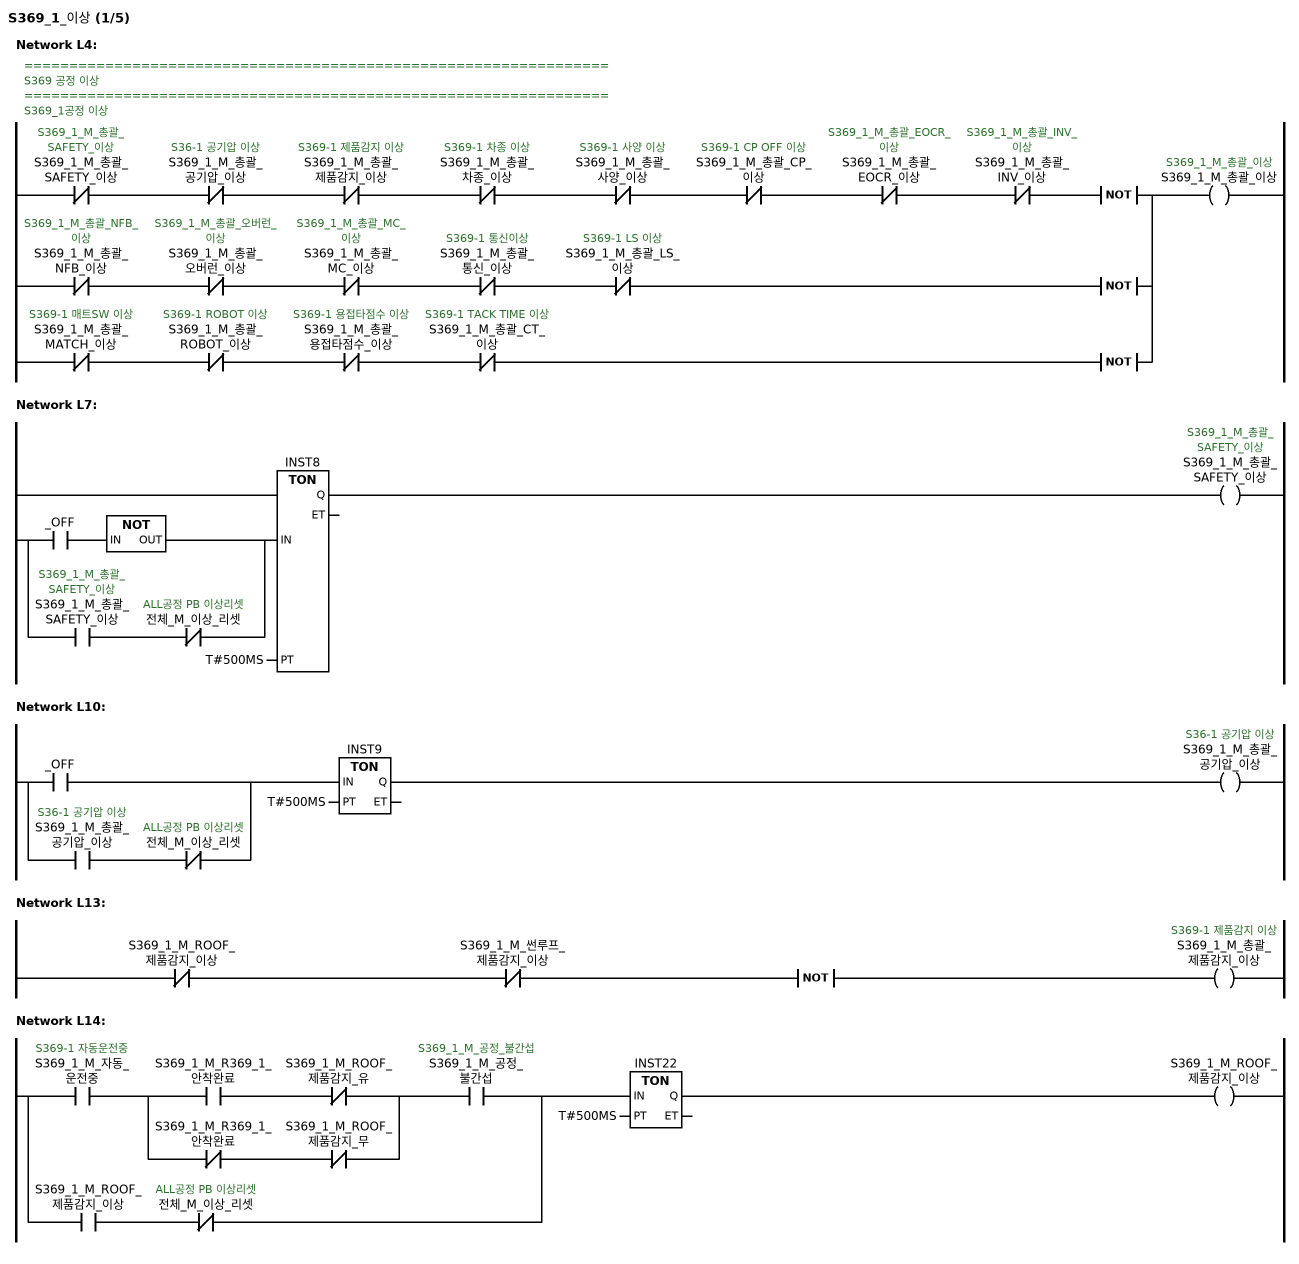
(* [picture p264: S369_1_이상 rungs L4-L14] *)
(* ================================================================= *)
(* S369 공정 이상 *)
(* ================================================================= *)
(* S369_1공정 이상 *)
(* Rung L4 *)
S369_1_M_총괄_이상 := NOT (NOT S369_1_M_총괄_SAFETY_이상 AND NOT S369_1_M_총괄_공기압_이상 AND NOT S369_1_M_총괄_제품감지_이상 AND NOT S369_1_M_총괄_차종_이상 AND NOT S369_1_M_총괄_사양_이상 AND NOT S369_1_M_총괄_CP_이상 AND NOT S369_1_M_총괄_EOCR_이상 AND NOT S369_1_M_총괄_INV_이상) OR NOT (NOT S369_1_M_총괄_NFB_이상 AND NOT S369_1_M_총괄_오버런_이상 AND NOT S369_1_M_총괄_MC_이상 AND NOT S369_1_M_총괄_통신_이상 AND NOT S369_1_M_총괄_LS_이상) OR NOT (NOT S369_1_M_총괄_MATCH_이상 AND NOT S369_1_M_총괄_ROBOT_이상 AND NOT S369_1_M_총괄_용접타점수_이상 AND NOT S369_1_M_총괄_CT_이상);
(* Rung L7 *)
INST8(IN := (NOT _OFF) OR (S369_1_M_총괄_SAFETY_이상 AND NOT 전체_M_이상_리셋), PT := T#500MS);
S369_1_M_총괄_SAFETY_이상 := INST8.Q;
(* Rung L10 *)
INST9(IN := _OFF OR (S369_1_M_총괄_공기압_이상 AND NOT 전체_M_이상_리셋), PT := T#500MS);
S369_1_M_총괄_공기압_이상 := INST9.Q;
(* Rung L13 *)
S369_1_M_총괄_제품감지_이상 := NOT (NOT S369_1_M_ROOF_제품감지_이상 AND NOT S369_1_M_썬루프_제품감지_이상);
(* Rung L14 *)
INST22(IN := (S369_1_M_자동_운전중 AND ((S369_1_M_R369_1_안착완료 AND NOT S369_1_M_ROOF_제품감지_유) OR (NOT S369_1_M_R369_1_안착완료 AND NOT S369_1_M_ROOF_제품감지_무)) AND S369_1_M_공정_불간섭) OR (S369_1_M_ROOF_제품감지_이상 AND NOT 전체_M_이상_리셋), PT := T#500MS);
S369_1_M_ROOF_제품감지_이상 := INST22.Q;

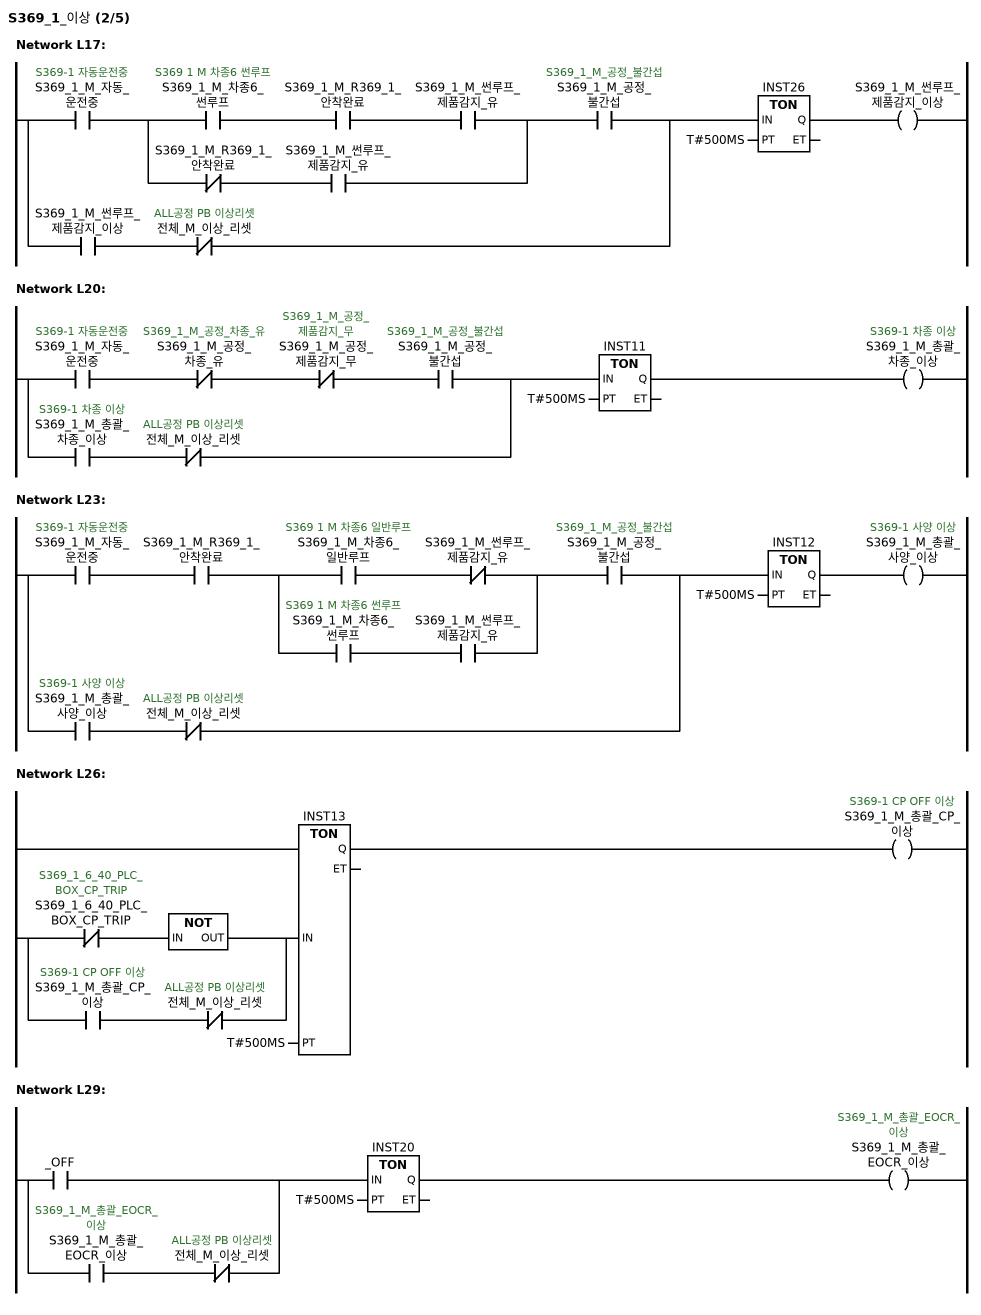
(* Rung L17 *)
INST26(IN := (S369_1_M_자동_운전중 AND ((S369_1_M_차종6_썬루프 AND S369_1_M_R369_1_안착완료 AND S369_1_M_썬루프_제품감지_유) OR (NOT S369_1_M_R369_1_안착완료 AND S369_1_M_썬루프_제품감지_유)) AND S369_1_M_공정_불간섭) OR (S369_1_M_썬루프_제품감지_이상 AND NOT 전체_M_이상_리셋), PT := T#500MS);
S369_1_M_썬루프_제품감지_이상 := INST26.Q;
(* Rung L20 *)
INST11(IN := (S369_1_M_자동_운전중 AND NOT S369_1_M_공정_차종_유 AND NOT S369_1_M_공정_제품감지_무 AND S369_1_M_공정_불간섭) OR (S369_1_M_총괄_차종_이상 AND NOT 전체_M_이상_리셋), PT := T#500MS);
S369_1_M_총괄_차종_이상 := INST11.Q;
(* Rung L23 *)
INST12(IN := (S369_1_M_자동_운전중 AND S369_1_M_R369_1_안착완료 AND ((S369_1_M_차종6_일반루프 AND NOT S369_1_M_썬루프_제품감지_유) OR (S369_1_M_차종6_썬루프 AND S369_1_M_썬루프_제품감지_유)) AND S369_1_M_공정_불간섭) OR (S369_1_M_총괄_사양_이상 AND NOT 전체_M_이상_리셋), PT := T#500MS);
S369_1_M_총괄_사양_이상 := INST12.Q;
(* Rung L26 *)
INST13(IN := (NOT (NOT S369_1_6_40_PLC_BOX_CP_TRIP)) OR (S369_1_M_총괄_CP_이상 AND NOT 전체_M_이상_리셋), PT := T#500MS);
S369_1_M_총괄_CP_이상 := INST13.Q;
(* Rung L29 *)
INST20(IN := _OFF OR (S369_1_M_총괄_EOCR_이상 AND NOT 전체_M_이상_리셋), PT := T#500MS);
S369_1_M_총괄_EOCR_이상 := INST20.Q;

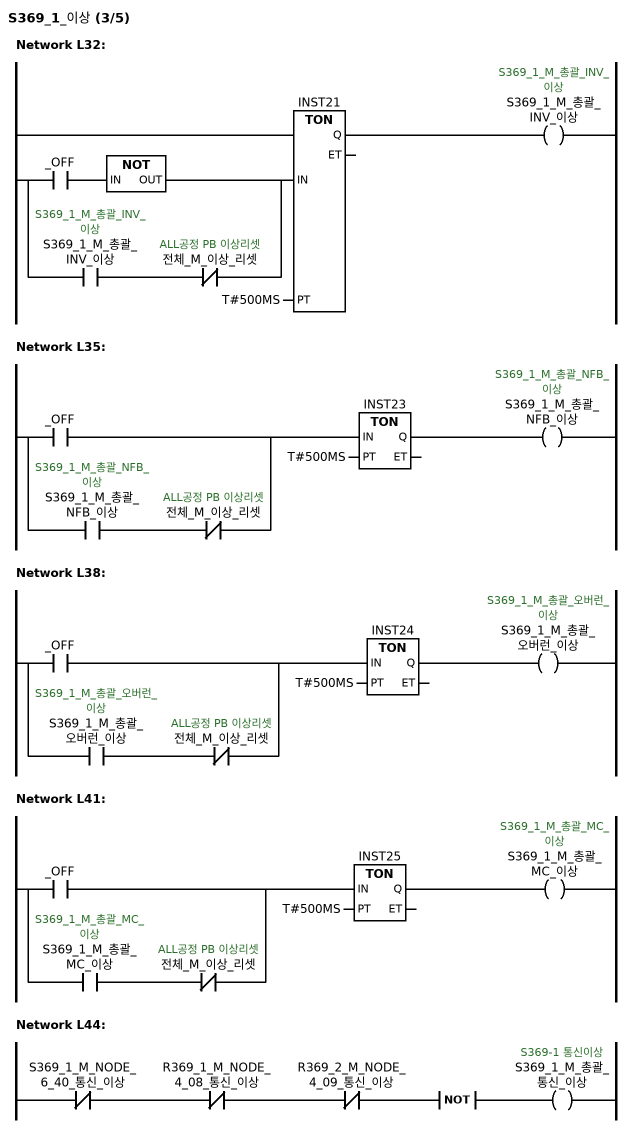
(* Rung L32 *)
INST21(IN := (NOT _OFF) OR (S369_1_M_총괄_INV_이상 AND NOT 전체_M_이상_리셋), PT := T#500MS);
S369_1_M_총괄_INV_이상 := INST21.Q;
(* Rung L35 *)
INST23(IN := _OFF OR (S369_1_M_총괄_NFB_이상 AND NOT 전체_M_이상_리셋), PT := T#500MS);
S369_1_M_총괄_NFB_이상 := INST23.Q;
(* Rung L38 *)
INST24(IN := _OFF OR (S369_1_M_총괄_오버런_이상 AND NOT 전체_M_이상_리셋), PT := T#500MS);
S369_1_M_총괄_오버런_이상 := INST24.Q;
(* Rung L41 *)
INST25(IN := _OFF OR (S369_1_M_총괄_MC_이상 AND NOT 전체_M_이상_리셋), PT := T#500MS);
S369_1_M_총괄_MC_이상 := INST25.Q;
(* Rung L44 *)
S369_1_M_총괄_통신_이상 := NOT (NOT S369_1_M_NODE_6_40_통신_이상 AND NOT R369_1_M_NODE_4_08_통신_이상 AND NOT R369_2_M_NODE_4_09_통신_이상);

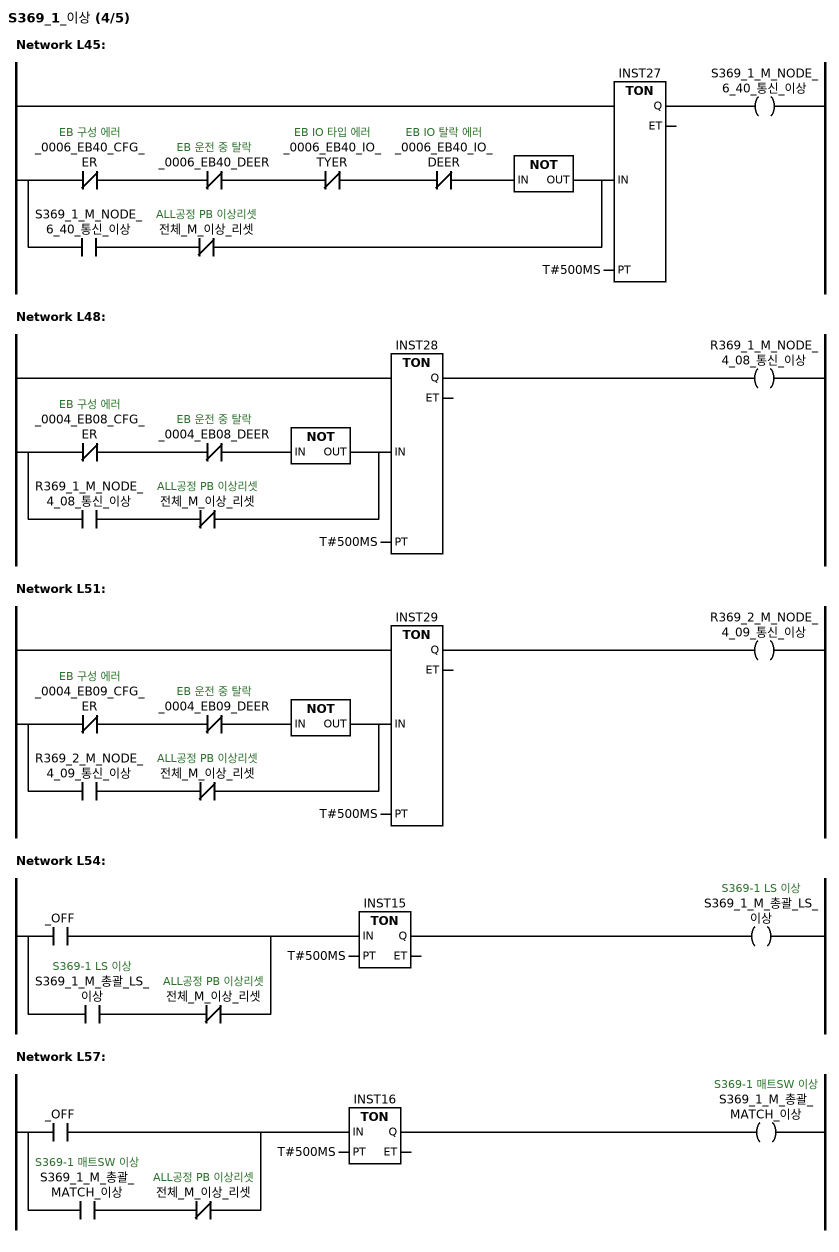
(* Rung L45 *)
INST27(IN := (NOT (NOT _0006_EB40_CFG_ER AND NOT _0006_EB40_DEER AND NOT _0006_EB40_IO_TYER AND NOT _0006_EB40_IO_DEER)) OR (S369_1_M_NODE_6_40_통신_이상 AND NOT 전체_M_이상_리셋), PT := T#500MS);
S369_1_M_NODE_6_40_통신_이상 := INST27.Q;
(* Rung L48 *)
INST28(IN := (NOT (NOT _0004_EB08_CFG_ER AND NOT _0004_EB08_DEER)) OR (R369_1_M_NODE_4_08_통신_이상 AND NOT 전체_M_이상_리셋), PT := T#500MS);
R369_1_M_NODE_4_08_통신_이상 := INST28.Q;
(* Rung L51 *)
INST29(IN := (NOT (NOT _0004_EB09_CFG_ER AND NOT _0004_EB09_DEER)) OR (R369_2_M_NODE_4_09_통신_이상 AND NOT 전체_M_이상_리셋), PT := T#500MS);
R369_2_M_NODE_4_09_통신_이상 := INST29.Q;
(* Rung L54 *)
INST15(IN := _OFF OR (S369_1_M_총괄_LS_이상 AND NOT 전체_M_이상_리셋), PT := T#500MS);
S369_1_M_총괄_LS_이상 := INST15.Q;
(* Rung L57 *)
INST16(IN := _OFF OR (S369_1_M_총괄_MATCH_이상 AND NOT 전체_M_이상_리셋), PT := T#500MS);
S369_1_M_총괄_MATCH_이상 := INST16.Q;

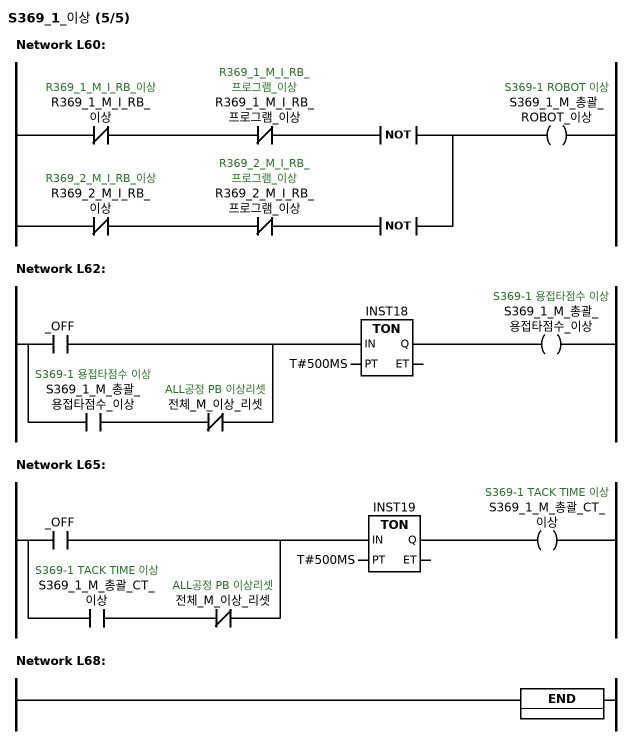
(* Rung L60 *)
S369_1_M_총괄_ROBOT_이상 := NOT (NOT R369_1_M_I_RB_이상 AND NOT R369_1_M_I_RB_프로그램_이상) OR NOT (NOT R369_2_M_I_RB_이상 AND NOT R369_2_M_I_RB_프로그램_이상);
(* Rung L62 *)
INST18(IN := _OFF OR (S369_1_M_총괄_용접타점수_이상 AND NOT 전체_M_이상_리셋), PT := T#500MS);
S369_1_M_총괄_용접타점수_이상 := INST18.Q;
(* Rung L65 *)
INST19(IN := _OFF OR (S369_1_M_총괄_CT_이상 AND NOT 전체_M_이상_리셋), PT := T#500MS);
S369_1_M_총괄_CT_이상 := INST19.Q;
(* Rung L68 *)
END();
END_PROGRAM

PROGRAM S369_유틸리티 (* task: 스캔 프로그램 *)
VAR_EXTERNAL RETAIN
    ALWAYS_OFF : BOOL; (* AT %MW3.0 *) (* 항시 OFF *)
    HMI_M_선택_MOD_S368 : BOOL; (* AT %MW6.6 *) (* HMI M 선택 MOD S368 *)
    HMI_M_선택_MOD_S369_LD : BOOL; (* AT %MW6.8 *) (* HMI M 선택 MOD S369 *)
    HMI_M_선택_MOD_S369_UD : BOOL; (* AT %MW6.9 *)
    S368_M_공정_제품감지_무 : BOOL; (* AT %MW4001.6 *) (* S368_M_공정_제품감지_무 *)
    S368_M_공정_차종_무 : BOOL; (* AT %MW4002.1 *) (* S368_M_공정_차종_무 *)
    S368_M_작업완료_SET_PLS : BOOL; (* AT %MW4000.8 *) (* S368 M 작업완료 SET PLS *)
    S368_M_작업완료_리셋_PLS : BOOL; (* AT %MW4000.9 *) (* S368 M 작업완료 리셋 PLS *)
    S369_1_M_공정_차종_무 : BOOL; (* AT %MW4502.1 *) (* S369_1_M_공정_차종_무 *)
    S369_1_M_공정_차종_유 : BOOL; (* AT %MW4502.0 *) (* S369_1_M_공정_차종_유 *)
    S369_1_M_총괄_이상 : BOOL; (* AT %MW4509.0 *) (* S369_1_M_총괄_이상 *)
    S369_M_LD_BYPASS_보조 : BOOL; (* AT %MW5003.14 *)
    S369_M_LD_EJECT_상승단 : BOOL; (* AT %MW5100.3 *) (* S369_M_LD_EJECT_상승단 *)
    S369_M_LD_EJECT_하강단 : BOOL; (* AT %MW5100.4 *) (* S369_M_LD_EJECT_하강단 *)
    S369_M_LD_LH_LAT_전진단 : BOOL; (* AT %MW5101.3 *) (* S369_M_LD_LH_LAT_전진단 *)
    S369_M_LD_LH_LAT_후진단 : BOOL; (* AT %MW5101.4 *) (* S369_M_LD_LH_LAT_후진단 *)
    S369_M_LD_RH_LAT_전진단 : BOOL; (* AT %MW5102.3 *) (* S369_M_LD_RH_LAT_전진단 *)
    S369_M_LD_RH_LAT_후진단 : BOOL; (* AT %MW5102.4 *) (* S369_M_LD_RH_LAT_후진단 *)
    S369_M_LD_작업완료_SET_PLS : BOOL; (* AT %MW5000.6 *)
    S369_M_LD_작업완료_리셋_PLS : BOOL; (* AT %MW5000.7 *)
    S369_M_R308_3_언로딩가능 : BOOL; (* AT %MW5004.9 *)
    S369_M_R308_3_언로딩완료 : BOOL; (* AT %MW5001.5 *)
    S369_M_R308_3_클램프완료 : BOOL; (* AT %MW5001.4 *)
    S369_M_R308_3_클램프요구 : BOOL; (* AT %MW5004.11 *)
    S369_M_R308_3_행거안착가능 : BOOL; (* AT %MW5004.10 *)
    S369_M_R308_3_행거안착완료 : BOOL; (* AT %MW5001.3 *)
    S369_M_R369_2_로딩가능 : BOOL; (* AT %MW5004.8 *)
    S369_M_R369_2_로딩완료 : BOOL; (* AT %MW5001.2 *)
    S369_M_UD_BYPASS_보조 : BOOL; (* AT %MW5003.15 *) (* S369 M BYPASS 보조 *)
    S369_M_UD_DOCK_CLP_전진단 : BOOL; (* AT %MW5111.3 *) (* S369_M_UD_DOCK_CLP_전진단 *)
    S369_M_UD_DOCK_CLP_후진단 : BOOL; (* AT %MW5111.4 *) (* S369_M_UD_DOCK_CLP_후진단 *)
    S369_M_UD_EJECT_상승단 : BOOL; (* AT %MW5108.3 *) (* S369_M_UD_EJECT_상승단 *)
    S369_M_UD_EJECT_하강단 : BOOL; (* AT %MW5108.4 *) (* S369_M_UD_EJECT_하강단 *)
    S369_M_UD_LH_LAT_전진단 : BOOL; (* AT %MW5109.3 *) (* S369_M_UD_LH_LAT_전진단 *)
    S369_M_UD_LH_LAT_후진단 : BOOL; (* AT %MW5109.4 *) (* S369_M_UD_LH_LAT_후진단 *)
    S369_M_UD_RH_LAT_전진단 : BOOL; (* AT %MW5110.3 *) (* S369_M_UD_RH_LAT_전진단 *)
    S369_M_UD_RH_LAT_후진단 : BOOL; (* AT %MW5110.4 *) (* S369_M_UD_RH_LAT_후진단 *)
    S369_M_UD_작업완료_SET_PLS : BOOL; (* AT %MW5000.8 *) (* S369 M 작업완료 SET PLS *)
    S369_M_UD_작업완료_리셋_PLS : BOOL; (* AT %MW5000.9 *) (* S369 M 작업완료 리셋 PLS *)
    S369_M_로딩_공정_불간섭 : BOOL; (* AT %MW5004.2 *) (* S369_M_공정_불간섭 *)
    S369_M_로딩_공정_원위치 : BOOL; (* AT %MW5004.0 *) (* S369_M_공정_원위치 *)
    S369_M_로딩_리셋보조 : BOOL; (* AT %MW5000.13 *)
    S369_M_로딩_이젝터_제품감지_무 : BOOL; (* AT %MW5001.9 *)
    S369_M_로딩_이젝터_제품감지_유 : BOOL; (* AT %MW5001.8 *)
    S369_M_로딩_작업_완료 : BOOL; (* AT %MW5001.0 *) (* S369_M_작업_완료 *)
    S369_M_로딩버퍼_SEQ : WORD; (* AT %MW10240 *) (* S369 M 로딩버퍼 SEQ *)
    S369_M_로딩버퍼_제품감지_무 : BOOL; (* AT %MW5005.1 *) (* S369_로딩버퍼_제품감지_무 *)
    S369_M_로딩버퍼_제품감지_유 : BOOL; (* AT %MW5005.0 *) (* S369_로딩버퍼_제품감지_유 *)
    S369_M_로딩버퍼_차종1_AX : BOOL; (* AT %MW10241.0 *) (* S369 M 로딩버퍼 차종1 AX *)
    S369_M_로딩버퍼_차종1_B : BOOL; (* AT %MW10241.1 *) (* S369 M 로딩버퍼 차종1 B *)
    S369_M_로딩버퍼_차종1_C : BOOL; (* AT %MW10241.2 *) (* S369 M 로딩버퍼 차종1 C *)
    S369_M_로딩버퍼_차종1_D : BOOL; (* AT %MW10241.3 *) (* S369 M 로딩버퍼 차종1 D *)
    S369_M_로딩버퍼_차종1_E : BOOL; (* AT %MW10241.4 *) (* S369 M 로딩버퍼 차종1 E *)
    S369_M_로딩버퍼_차종1_F : BOOL; (* AT %MW10241.5 *) (* S369 M 로딩버퍼 차종1 F *)
    S369_M_로딩버퍼_차종1_G : BOOL; (* AT %MW10241.6 *) (* S369 M 로딩버퍼 차종1 G *)
    S369_M_로딩버퍼_차종1_H : BOOL; (* AT %MW10241.7 *) (* S369 M 로딩버퍼 차종1 H *)
    S369_M_로딩버퍼_차종2_3DR : BOOL; (* AT %MW10241.8 *) (* S369 M 로딩버퍼 차종2 3DR *)
    S369_M_로딩버퍼_차종2_4DR : BOOL; (* AT %MW10241.9 *) (* S369 M 로딩버퍼 차종2 4DR *)
    S369_M_로딩버퍼_차종2_5DR : BOOL; (* AT %MW10241.10 *) (* S369 M 로딩버퍼 차종2 5DR *)
    S369_M_로딩버퍼_차종2_SP1 : BOOL; (* AT %MW10241.12 *) (* S369 M 로딩버퍼 차종2 SP1 *)
    S369_M_로딩버퍼_차종2_SP2 : BOOL; (* AT %MW10241.13 *) (* S369 M 로딩버퍼 차종2 SP2 *)
    S369_M_로딩버퍼_차종2_WGN : BOOL; (* AT %MW10241.11 *) (* S369 M 로딩버퍼 차종2 WGN *)
    S369_M_로딩버퍼_차종3_LHD : BOOL; (* AT %MW10241.14 *) (* S369 M 로딩버퍼 차종3 LHD *)
    S369_M_로딩버퍼_차종3_RHD : BOOL; (* AT %MW10241.15 *) (* S369 M 로딩버퍼 차종3 RHD *)
    S369_M_로딩버퍼_차종4_EEC : BOOL; (* AT %MW10242.3 *) (* S369 M 로딩버퍼 차종4 EEC *)
    S369_M_로딩버퍼_차종4_SP1 : BOOL; (* AT %MW10242.8 *) (* S369 M 로딩버퍼 차종4 SP1 *)
    S369_M_로딩버퍼_차종4_SP2 : BOOL; (* AT %MW10242.9 *) (* S369 M 로딩버퍼 차종4 SP2 *)
    S369_M_로딩버퍼_차종4_SP3 : BOOL; (* AT %MW10242.11 *) (* S369 M 로딩버퍼 차종4 SP3 *)
    S369_M_로딩버퍼_차종4_SP4 : BOOL; (* AT %MW10242.12 *) (* S369 M 로딩버퍼 차종4 SP4 *)
    S369_M_로딩버퍼_차종4_SP5 : BOOL; (* AT %MW10242.13 *) (* S369 M 로딩버퍼 차종4 SP5 *)
    S369_M_로딩버퍼_차종4_SP6 : BOOL; (* AT %MW10242.14 *) (* S369 M 로딩버퍼 차종4 SP6 *)
    S369_M_로딩버퍼_차종4_SP7 : BOOL; (* AT %MW10242.15 *) (* S369 M 로딩버퍼 차종4 SP7 *)
    S369_M_로딩버퍼_차종4_내수 : BOOL; (* AT %MW10242.0 *) (* S369 M 로딩버퍼 차종4 내수 *)
    S369_M_로딩버퍼_차종4_러시아 : BOOL; (* AT %MW10242.10 *) (* S369 M 로딩버퍼 차종4 러시아 *)
    S369_M_로딩버퍼_차종4_북미 : BOOL; (* AT %MW10242.2 *) (* S369 M 로딩버퍼 차종4 북미 *)
    S369_M_로딩버퍼_차종4_브라질 : BOOL; (* AT %MW10242.7 *) (* S369 M 로딩버퍼 차종4 브라질 *)
    S369_M_로딩버퍼_차종4_수출 : BOOL; (* AT %MW10242.1 *) (* S369 M 로딩버퍼 차종4 수출 *)
    S369_M_로딩버퍼_차종4_중국 : BOOL; (* AT %MW10242.6 *) (* S369 M 로딩버퍼 차종4 중국 *)
    S369_M_로딩버퍼_차종4_중동 : BOOL; (* AT %MW10242.5 *) (* S369 M 로딩버퍼 차종4 중동 *)
    S369_M_로딩버퍼_차종4_호주 : BOOL; (* AT %MW10242.4 *) (* S369 M 로딩버퍼 차종4 호주 *)
    S369_M_로딩버퍼_차종5_AT : BOOL; (* AT %MW10243.1 *) (* S369 M 로딩버퍼 차종5 AT *)
    S369_M_로딩버퍼_차종5_MT : BOOL; (* AT %MW10243.0 *) (* S369 M 로딩버퍼 차종5 MT *)
    S369_M_로딩버퍼_차종5_SP1 : BOOL; (* AT %MW10243.2 *) (* S369 M 로딩버퍼 차종5 SP1 *)
    S369_M_로딩버퍼_차종6_DSROOF : BOOL; (* AT %MW10243.6 *) (* S369 M 로딩버퍼 차종6 DSROOF *)
    S369_M_로딩버퍼_차종6_SP1 : BOOL; (* AT %MW10243.7 *) (* S369 M 로딩버퍼 차종6 SP1 *)
    S369_M_로딩버퍼_차종6_썬루프 : BOOL; (* AT %MW10243.4 *) (* S369 M 로딩버퍼 차종6 썬루프 *)
    S369_M_로딩버퍼_차종6_일반루프 : BOOL; (* AT %MW10243.3 *) (* S369 M 로딩버퍼 차종6 일반루프 *)
    S369_M_로딩버퍼_차종6_파노라마루프 : BOOL; (* AT %MW10243.5 *) (* S369 M 로딩버퍼 차종6 파노라마루프 *)
    S369_M_로딩버퍼_차종7_DSL : BOOL; (* AT %MW10243.9 *) (* S369 M 로딩버퍼 차종7 DSL *)
    S369_M_로딩버퍼_차종7_GSL : BOOL; (* AT %MW10243.8 *) (* S369 M 로딩버퍼 차종7 GSL *)
    S369_M_로딩버퍼_차종7_SP1 : BOOL; (* AT %MW10243.10 *) (* S369 M 로딩버퍼 차종7 SP1 *)
    S369_M_로딩버퍼_차종7_SP2 : BOOL; (* AT %MW10243.11 *) (* S369 M 로딩버퍼 차종7 SP2 *)
    S369_M_로딩버퍼_차종7_SP3 : BOOL; (* AT %MW10243.12 *) (* S369 M 로딩버퍼 차종7 SP3 *)
    S369_M_로딩버퍼_차종7_SP4 : BOOL; (* AT %MW10243.13 *) (* S369 M 로딩버퍼 차종7 SP4 *)
    S369_M_로딩버퍼_차종7_SP5 : BOOL; (* AT %MW10243.14 *) (* S369 M 로딩버퍼 차종7 SP5 *)
    S369_M_로딩버퍼_차종7_SP6 : BOOL; (* AT %MW10243.15 *) (* S369 M 로딩버퍼 차종7 SP6 *)
    S369_M_로딩버퍼_차종8_2WD : BOOL; (* AT %MW10244.0 *) (* S369 M 로딩버퍼 차종8 2WD *)
    S369_M_로딩버퍼_차종8_4WD : BOOL; (* AT %MW10244.1 *) (* S369 M 로딩버퍼 차종8 4WD *)
    S369_M_로딩버퍼_차종8_SP1 : BOOL; (* AT %MW10244.2 *) (* S369 M 로딩버퍼 차종8 SP1 *)
    S369_M_로딩버퍼_차종9_MPI : BOOL; (* AT %MW10244.3 *) (* S369 M 로딩버퍼 차종9 MPI *)
    S369_M_로딩버퍼_차종9_SP1 : BOOL; (* AT %MW10244.5 *) (* S369 M 로딩버퍼 차종9 SP1 *)
    S369_M_로딩버퍼_차종9_SP10 : BOOL; (* AT %MW10244.14 *) (* S369 M 로딩버퍼 차종9 SP10 *)
    S369_M_로딩버퍼_차종9_SP11 : BOOL; (* AT %MW10244.15 *) (* S369 M 로딩버퍼 차종9 SP11 *)
    S369_M_로딩버퍼_차종9_SP2 : BOOL; (* AT %MW10244.6 *) (* S369 M 로딩버퍼 차종9 SP2 *)
    S369_M_로딩버퍼_차종9_SP3 : BOOL; (* AT %MW10244.7 *) (* S369 M 로딩버퍼 차종9 SP3 *)
    S369_M_로딩버퍼_차종9_SP4 : BOOL; (* AT %MW10244.8 *) (* S369 M 로딩버퍼 차종9 SP4 *)
    S369_M_로딩버퍼_차종9_SP5 : BOOL; (* AT %MW10244.9 *) (* S369 M 로딩버퍼 차종9 SP5 *)
    S369_M_로딩버퍼_차종9_SP6 : BOOL; (* AT %MW10244.10 *) (* S369 M 로딩버퍼 차종9 SP6 *)
    S369_M_로딩버퍼_차종9_SP7 : BOOL; (* AT %MW10244.11 *) (* S369 M 로딩버퍼 차종9 SP7 *)
    S369_M_로딩버퍼_차종9_SP8 : BOOL; (* AT %MW10244.12 *) (* S369 M 로딩버퍼 차종9 SP8 *)
    S369_M_로딩버퍼_차종9_SP9 : BOOL; (* AT %MW10244.13 *) (* S369 M 로딩버퍼 차종9 SP9 *)
    S369_M_로딩버퍼_차종9_T_GDI : BOOL; (* AT %MW10244.4 *) (* S369 M 로딩버퍼 차종9 T GDI *)
    S369_M_로딩버퍼_차종_OPT1_R_RACK_무 : BOOL; (* AT %MW10245.3 *) (* S369 M 로딩버퍼 차종 OPT1 R RACK 무 *)
    S369_M_로딩버퍼_차종_OPT1_R_RACK_유 : BOOL; (* AT %MW10245.2 *) (* S369 M 로딩버퍼 차종 OPT1 R RACK 유 *)
    S369_M_로딩버퍼_차종_OPT1_S_REP_EATER_무 : BOOL; (* AT %MW10245.7 *) (* S369 M 로딩버퍼 차종 OPT1 S REP EATER 무 *)
    S369_M_로딩버퍼_차종_OPT1_S_REP_EATER_유 : BOOL; (* AT %MW10245.6 *) (* S369 M 로딩버퍼 차종 OPT1 S REP EATER 유 *)
    S369_M_로딩버퍼_차종_OPT1_VAN_무 : BOOL; (* AT %MW10245.9 *) (* S369 M 로딩버퍼 차종 OPT1 VAN 무 *)
    S369_M_로딩버퍼_차종_OPT1_VAN_유 : BOOL; (* AT %MW10245.8 *) (* S369 M 로딩버퍼 차종 OPT1 VAN 유 *)
    S369_M_로딩버퍼_차종_OPT1_슬라이딩_무 : BOOL; (* AT %MW10245.1 *) (* S369 M 로딩버퍼 차종 OPT1 슬라이딩 무 *)
    S369_M_로딩버퍼_차종_OPT1_슬라이딩_유 : BOOL; (* AT %MW10245.0 *) (* S369 M 로딩버퍼 차종 OPT1 슬라이딩 유 *)
    S369_M_로딩버퍼_차종_OPT1_폴딩_무 : BOOL; (* AT %MW10245.5 *) (* S369 M 로딩버퍼 차종 OPT1 폴딩 무 *)
    S369_M_로딩버퍼_차종_OPT1_폴딩_유 : BOOL; (* AT %MW10245.4 *) (* S369 M 로딩버퍼 차종 OPT1 폴딩 유 *)
    S369_M_로딩버퍼_차종_공대차 : BOOL; (* AT %MW10250.12 *) (* S369 M 로딩버퍼 차종 공대차 *)
    S369_M_로딩버퍼_차종_공차 : BOOL; (* AT %MW10250.10 *) (* S369 M 로딩버퍼 차종 공차 *)
    S369_M_로딩버퍼_차종_무 : BOOL; (* AT %MW5002.1 *)
    S369_M_로딩버퍼_차종_불량차 : BOOL; (* AT %MW10250.11 *) (* S369 M 로딩버퍼 차종 불량차 *)
    S369_M_로딩버퍼_차종_유 : BOOL; (* AT %MW5002.0 *)
    S369_M_수동모드 : BOOL; (* AT %MW5000.3 *) (* S369 선택 수동모드 *)
    S369_M_언로딩_공정_불간섭 : BOOL; (* AT %MW5004.3 *)
    S369_M_언로딩_공정_원위치 : BOOL; (* AT %MW5004.1 *)
    S369_M_언로딩_이젝터_제품감지_무 : BOOL; (* AT %MW5001.11 *)
    S369_M_언로딩_이젝터_제품감지_유 : BOOL; (* AT %MW5001.10 *)
    S369_M_언로딩_작업_완료 : BOOL; (* AT %MW5001.1 *)
    S369_M_언로딩버퍼_SEQ : WORD; (* AT %MW10340 *) (* S369 M 언로딩버퍼 SEQ *)
    S369_M_언로딩버퍼_제품감지_무 : BOOL; (* AT %MW5005.11 *) (* S369_언로딩버퍼_제품감지_무 *)
    S369_M_언로딩버퍼_제품감지_유 : BOOL; (* AT %MW5005.10 *) (* S369_언로딩버퍼_제품감지_유 *)
    S369_M_언로딩버퍼_차종1_AX : BOOL; (* AT %MW10341.0 *) (* S369 M 언로딩버퍼 차종1 AX *)
    S369_M_언로딩버퍼_차종1_B : BOOL; (* AT %MW10341.1 *) (* S369 M 언로딩버퍼 차종1 B *)
    S369_M_언로딩버퍼_차종1_C : BOOL; (* AT %MW10341.2 *) (* S369 M 언로딩버퍼 차종1 C *)
    S369_M_언로딩버퍼_차종1_D : BOOL; (* AT %MW10341.3 *) (* S369 M 언로딩버퍼 차종1 D *)
    S369_M_언로딩버퍼_차종1_E : BOOL; (* AT %MW10341.4 *) (* S369 M 언로딩버퍼 차종1 E *)
    S369_M_언로딩버퍼_차종1_F : BOOL; (* AT %MW10341.5 *) (* S369 M 언로딩버퍼 차종1 F *)
    S369_M_언로딩버퍼_차종1_G : BOOL; (* AT %MW10341.6 *) (* S369 M 언로딩버퍼 차종1 G *)
    S369_M_언로딩버퍼_차종1_H : BOOL; (* AT %MW10341.7 *) (* S369 M 언로딩버퍼 차종1 H *)
    S369_M_언로딩버퍼_차종2_3DR : BOOL; (* AT %MW10341.8 *) (* S369 M 언로딩버퍼 차종2 3DR *)
    S369_M_언로딩버퍼_차종2_4DR : BOOL; (* AT %MW10341.9 *) (* S369 M 언로딩버퍼 차종2 4DR *)
    S369_M_언로딩버퍼_차종2_5DR : BOOL; (* AT %MW10341.10 *) (* S369 M 언로딩버퍼 차종2 5DR *)
    S369_M_언로딩버퍼_차종2_SP1 : BOOL; (* AT %MW10341.12 *) (* S369 M 언로딩버퍼 차종2 SP1 *)
    S369_M_언로딩버퍼_차종2_SP2 : BOOL; (* AT %MW10341.13 *) (* S369 M 언로딩버퍼 차종2 SP2 *)
    S369_M_언로딩버퍼_차종2_WGN : BOOL; (* AT %MW10341.11 *) (* S369 M 언로딩버퍼 차종2 WGN *)
    S369_M_언로딩버퍼_차종3_LHD : BOOL; (* AT %MW10341.14 *) (* S369 M 언로딩버퍼 차종3 LHD *)
    S369_M_언로딩버퍼_차종3_RHD : BOOL; (* AT %MW10341.15 *) (* S369 M 언로딩버퍼 차종3 RHD *)
    S369_M_언로딩버퍼_차종4_EEC : BOOL; (* AT %MW10342.3 *) (* S369 M 언로딩버퍼 차종4 EEC *)
    S369_M_언로딩버퍼_차종4_SP1 : BOOL; (* AT %MW10342.8 *) (* S369 M 언로딩버퍼 차종4 SP1 *)
    S369_M_언로딩버퍼_차종4_SP2 : BOOL; (* AT %MW10342.9 *) (* S369 M 언로딩버퍼 차종4 SP2 *)
    S369_M_언로딩버퍼_차종4_SP3 : BOOL; (* AT %MW10342.11 *) (* S369 M 언로딩버퍼 차종4 SP3 *)
    S369_M_언로딩버퍼_차종4_SP4 : BOOL; (* AT %MW10342.12 *) (* S369 M 언로딩버퍼 차종4 SP4 *)
    S369_M_언로딩버퍼_차종4_SP5 : BOOL; (* AT %MW10342.13 *) (* S369 M 언로딩버퍼 차종4 SP5 *)
    S369_M_언로딩버퍼_차종4_SP6 : BOOL; (* AT %MW10342.14 *) (* S369 M 언로딩버퍼 차종4 SP6 *)
    S369_M_언로딩버퍼_차종4_SP7 : BOOL; (* AT %MW10342.15 *) (* S369 M 언로딩버퍼 차종4 SP7 *)
    S369_M_언로딩버퍼_차종4_내수 : BOOL; (* AT %MW10342.0 *) (* S369 M 언로딩버퍼 차종4 내수 *)
    S369_M_언로딩버퍼_차종4_러시아 : BOOL; (* AT %MW10342.10 *) (* S369 M 언로딩버퍼 차종4 러시아 *)
    S369_M_언로딩버퍼_차종4_북미 : BOOL; (* AT %MW10342.2 *) (* S369 M 언로딩버퍼 차종4 북미 *)
    S369_M_언로딩버퍼_차종4_브라질 : BOOL; (* AT %MW10342.7 *) (* S369 M 언로딩버퍼 차종4 브라질 *)
    S369_M_언로딩버퍼_차종4_수출 : BOOL; (* AT %MW10342.1 *) (* S369 M 언로딩버퍼 차종4 수출 *)
    S369_M_언로딩버퍼_차종4_중국 : BOOL; (* AT %MW10342.6 *) (* S369 M 언로딩버퍼 차종4 중국 *)
    S369_M_언로딩버퍼_차종4_중동 : BOOL; (* AT %MW10342.5 *) (* S369 M 언로딩버퍼 차종4 중동 *)
    S369_M_언로딩버퍼_차종4_호주 : BOOL; (* AT %MW10342.4 *) (* S369 M 언로딩버퍼 차종4 호주 *)
    S369_M_언로딩버퍼_차종5_AT : BOOL; (* AT %MW10343.1 *) (* S369 M 언로딩버퍼 차종5 AT *)
    S369_M_언로딩버퍼_차종5_MT : BOOL; (* AT %MW10343.0 *) (* S369 M 언로딩버퍼 차종5 MT *)
    S369_M_언로딩버퍼_차종5_SP1 : BOOL; (* AT %MW10343.2 *) (* S369 M 언로딩버퍼 차종5 SP1 *)
    S369_M_언로딩버퍼_차종6_DSROOF : BOOL; (* AT %MW10343.6 *) (* S369 M 언로딩버퍼 차종6 DSROOF *)
    S369_M_언로딩버퍼_차종6_SP1 : BOOL; (* AT %MW10343.7 *) (* S369 M 언로딩버퍼 차종6 SP1 *)
    S369_M_언로딩버퍼_차종6_썬루프 : BOOL; (* AT %MW10343.4 *) (* S369 M 언로딩버퍼 차종6 썬루프 *)
    S369_M_언로딩버퍼_차종6_일반루프 : BOOL; (* AT %MW10343.3 *) (* S369 M 언로딩버퍼 차종6 일반루프 *)
    S369_M_언로딩버퍼_차종6_파노라마루프 : BOOL; (* AT %MW10343.5 *) (* S369 M 언로딩버퍼 차종6 파노라마루프 *)
    S369_M_언로딩버퍼_차종7_DSL : BOOL; (* AT %MW10343.9 *) (* S369 M 언로딩버퍼 차종7 DSL *)
    S369_M_언로딩버퍼_차종7_GSL : BOOL; (* AT %MW10343.8 *) (* S369 M 언로딩버퍼 차종7 GSL *)
    S369_M_언로딩버퍼_차종7_SP1 : BOOL; (* AT %MW10343.10 *) (* S369 M 언로딩버퍼 차종7 SP1 *)
    S369_M_언로딩버퍼_차종7_SP2 : BOOL; (* AT %MW10343.11 *) (* S369 M 언로딩버퍼 차종7 SP2 *)
    S369_M_언로딩버퍼_차종7_SP3 : BOOL; (* AT %MW10343.12 *) (* S369 M 언로딩버퍼 차종7 SP3 *)
    S369_M_언로딩버퍼_차종7_SP4 : BOOL; (* AT %MW10343.13 *) (* S369 M 언로딩버퍼 차종7 SP4 *)
    S369_M_언로딩버퍼_차종7_SP5 : BOOL; (* AT %MW10343.14 *) (* S369 M 언로딩버퍼 차종7 SP5 *)
    S369_M_언로딩버퍼_차종7_SP6 : BOOL; (* AT %MW10343.15 *) (* S369 M 언로딩버퍼 차종7 SP6 *)
    S369_M_언로딩버퍼_차종8_2WD : BOOL; (* AT %MW10344.0 *) (* S369 M 언로딩버퍼 차종8 2WD *)
    S369_M_언로딩버퍼_차종8_4WD : BOOL; (* AT %MW10344.1 *) (* S369 M 언로딩버퍼 차종8 4WD *)
    S369_M_언로딩버퍼_차종8_SP1 : BOOL; (* AT %MW10344.2 *) (* S369 M 언로딩버퍼 차종8 SP1 *)
    S369_M_언로딩버퍼_차종9_MPI : BOOL; (* AT %MW10344.3 *) (* S369 M 언로딩버퍼 차종9 MPI *)
    S369_M_언로딩버퍼_차종9_SP1 : BOOL; (* AT %MW10344.5 *) (* S369 M 언로딩버퍼 차종9 SP1 *)
    S369_M_언로딩버퍼_차종9_SP10 : BOOL; (* AT %MW10344.14 *) (* S369 M 언로딩버퍼 차종9 SP10 *)
    S369_M_언로딩버퍼_차종9_SP11 : BOOL; (* AT %MW10344.15 *) (* S369 M 언로딩버퍼 차종9 SP11 *)
    S369_M_언로딩버퍼_차종9_SP2 : BOOL; (* AT %MW10344.6 *) (* S369 M 언로딩버퍼 차종9 SP2 *)
    S369_M_언로딩버퍼_차종9_SP3 : BOOL; (* AT %MW10344.7 *) (* S369 M 언로딩버퍼 차종9 SP3 *)
    S369_M_언로딩버퍼_차종9_SP4 : BOOL; (* AT %MW10344.8 *) (* S369 M 언로딩버퍼 차종9 SP4 *)
    S369_M_언로딩버퍼_차종9_SP5 : BOOL; (* AT %MW10344.9 *) (* S369 M 언로딩버퍼 차종9 SP5 *)
    S369_M_언로딩버퍼_차종9_SP6 : BOOL; (* AT %MW10344.10 *) (* S369 M 언로딩버퍼 차종9 SP6 *)
    S369_M_언로딩버퍼_차종9_SP7 : BOOL; (* AT %MW10344.11 *) (* S369 M 언로딩버퍼 차종9 SP7 *)
    S369_M_언로딩버퍼_차종9_SP8 : BOOL; (* AT %MW10344.12 *) (* S369 M 언로딩버퍼 차종9 SP8 *)
    S369_M_언로딩버퍼_차종9_SP9 : BOOL; (* AT %MW10344.13 *) (* S369 M 언로딩버퍼 차종9 SP9 *)
    S369_M_언로딩버퍼_차종9_T_GDI : BOOL; (* AT %MW10344.4 *) (* S369 M 언로딩버퍼 차종9 T GDI *)
    S369_M_언로딩버퍼_차종_OPT1_R_RACK_무 : BOOL; (* AT %MW10345.3 *) (* S369 M 언로딩버퍼 차종 OPT1 R RACK 무 *)
    S369_M_언로딩버퍼_차종_OPT1_R_RACK_유 : BOOL; (* AT %MW10345.2 *) (* S369 M 언로딩버퍼 차종 OPT1 R RACK 유 *)
    S369_M_언로딩버퍼_차종_OPT1_S_REP_EATER_무 : BOOL; (* AT %MW10345.7 *) (* S369 M 언로딩버퍼 차종 OPT1 S REP EATER 무 *)
    S369_M_언로딩버퍼_차종_OPT1_S_REP_EATER_유 : BOOL; (* AT %MW10345.6 *) (* S369 M 언로딩버퍼 차종 OPT1 S REP EATER 유 *)
    S369_M_언로딩버퍼_차종_OPT1_VAN_무 : BOOL; (* AT %MW10345.9 *) (* S369 M 언로딩버퍼 차종 OPT1 VAN 무 *)
    S369_M_언로딩버퍼_차종_OPT1_VAN_유 : BOOL; (* AT %MW10345.8 *) (* S369 M 언로딩버퍼 차종 OPT1 VAN 유 *)
    S369_M_언로딩버퍼_차종_OPT1_슬라이딩_무 : BOOL; (* AT %MW10345.1 *) (* S369 M 언로딩버퍼 차종 OPT1 슬라이딩 무 *)
    S369_M_언로딩버퍼_차종_OPT1_슬라이딩_유 : BOOL; (* AT %MW10345.0 *) (* S369 M 언로딩버퍼 차종 OPT1 슬라이딩 유 *)
    S369_M_언로딩버퍼_차종_OPT1_폴딩_무 : BOOL; (* AT %MW10345.5 *) (* S369 M 언로딩버퍼 차종 OPT1 폴딩 무 *)
    S369_M_언로딩버퍼_차종_OPT1_폴딩_유 : BOOL; (* AT %MW10345.4 *) (* S369 M 언로딩버퍼 차종 OPT1 폴딩 유 *)
    S369_M_언로딩버퍼_차종_공대차 : BOOL; (* AT %MW10350.12 *) (* S369 M 언로딩버퍼 차종 공대차 *)
    S369_M_언로딩버퍼_차종_공차 : BOOL; (* AT %MW10350.10 *) (* S369 M 언로딩버퍼 차종 공차 *)
    S369_M_언로딩버퍼_차종_무 : BOOL; (* AT %MW5002.3 *)
    S369_M_언로딩버퍼_차종_불량차 : BOOL; (* AT %MW10350.11 *) (* S369 M 언로딩버퍼 차종 불량차 *)
    S369_M_언로딩버퍼_차종_유 : BOOL; (* AT %MW5002.2 *)
    S369_M_운전준비_ON : BOOL; (* AT %MW5000.0 *) (* S369 운전준비 ON *)
    S369_M_이송버퍼01_제품감지_무 : BOOL; (* AT %MW5005.9 *) (* S369_이송버퍼01_제품감지_OFF *)
    S369_M_이송버퍼01_제품감지_유 : BOOL; (* AT %MW5005.8 *) (* S369_이송버퍼01_제품감지_ON *)
    S369_M_이송버퍼02_제품감지_무 : BOOL; (* AT %MW5005.7 *) (* S369_이송버퍼02_제품감지_OFF *)
    S369_M_이송버퍼02_제품감지_유 : BOOL; (* AT %MW5005.6 *) (* S369_이송버퍼02_제품감지_ON *)
    S369_M_이송버퍼03_제품감지_무 : BOOL; (* AT %MW5005.5 *) (* S369_이송버퍼03_제품감지_OFF *)
    S369_M_이송버퍼03_제품감지_유 : BOOL; (* AT %MW5005.4 *) (* S369_이송버퍼03_제품감지_ON *)
    S369_M_이송버퍼04_제품감지_무 : BOOL; (* AT %MW5005.3 *) (* S369_이송버퍼04_제품감지_OFF *)
    S369_M_이송버퍼04_제품감지_유 : BOOL; (* AT %MW5005.2 *) (* S369_이송버퍼04_제품감지_ON *)
    S369_M_이송버퍼1_SEQ : WORD; (* AT %MW10320 *) (* S369 M 이송버퍼1 SEQ *)
    S369_M_이송버퍼1_차종1_AX : BOOL; (* AT %MW10321.0 *) (* S369 M 이송버퍼1 차종1 AX *)
    S369_M_이송버퍼1_차종1_B : BOOL; (* AT %MW10321.1 *) (* S369 M 이송버퍼1 차종1 B *)
    S369_M_이송버퍼1_차종1_C : BOOL; (* AT %MW10321.2 *) (* S369 M 이송버퍼1 차종1 C *)
    S369_M_이송버퍼1_차종1_D : BOOL; (* AT %MW10321.3 *) (* S369 M 이송버퍼1 차종1 D *)
    S369_M_이송버퍼1_차종1_E : BOOL; (* AT %MW10321.4 *) (* S369 M 이송버퍼1 차종1 E *)
    S369_M_이송버퍼1_차종1_F : BOOL; (* AT %MW10321.5 *) (* S369 M 이송버퍼1 차종1 F *)
    S369_M_이송버퍼1_차종1_G : BOOL; (* AT %MW10321.6 *) (* S369 M 이송버퍼1 차종1 G *)
    S369_M_이송버퍼1_차종1_H : BOOL; (* AT %MW10321.7 *) (* S369 M 이송버퍼1 차종1 H *)
    S369_M_이송버퍼1_차종2_3DR : BOOL; (* AT %MW10321.8 *) (* S369 M 이송버퍼1 차종2 3DR *)
    S369_M_이송버퍼1_차종2_4DR : BOOL; (* AT %MW10321.9 *) (* S369 M 이송버퍼1 차종2 4DR *)
    S369_M_이송버퍼1_차종2_5DR : BOOL; (* AT %MW10321.10 *) (* S369 M 이송버퍼1 차종2 5DR *)
    S369_M_이송버퍼1_차종2_SP1 : BOOL; (* AT %MW10321.12 *) (* S369 M 이송버퍼1 차종2 SP1 *)
    S369_M_이송버퍼1_차종2_SP2 : BOOL; (* AT %MW10321.13 *) (* S369 M 이송버퍼1 차종2 SP2 *)
    S369_M_이송버퍼1_차종2_WGN : BOOL; (* AT %MW10321.11 *) (* S369 M 이송버퍼1 차종2 WGN *)
    S369_M_이송버퍼1_차종3_LHD : BOOL; (* AT %MW10321.14 *) (* S369 M 이송버퍼1 차종3 LHD *)
    S369_M_이송버퍼1_차종3_RHD : BOOL; (* AT %MW10321.15 *) (* S369 M 이송버퍼1 차종3 RHD *)
    S369_M_이송버퍼1_차종4_EEC : BOOL; (* AT %MW10322.3 *) (* S369 M 이송버퍼1 차종4 EEC *)
    S369_M_이송버퍼1_차종4_SP1 : BOOL; (* AT %MW10322.8 *) (* S369 M 이송버퍼1 차종4 SP1 *)
    S369_M_이송버퍼1_차종4_SP2 : BOOL; (* AT %MW10322.9 *) (* S369 M 이송버퍼1 차종4 SP2 *)
    S369_M_이송버퍼1_차종4_SP3 : BOOL; (* AT %MW10322.11 *) (* S369 M 이송버퍼1 차종4 SP3 *)
    S369_M_이송버퍼1_차종4_SP4 : BOOL; (* AT %MW10322.12 *) (* S369 M 이송버퍼1 차종4 SP4 *)
    S369_M_이송버퍼1_차종4_SP5 : BOOL; (* AT %MW10322.13 *) (* S369 M 이송버퍼1 차종4 SP5 *)
    S369_M_이송버퍼1_차종4_SP6 : BOOL; (* AT %MW10322.14 *) (* S369 M 이송버퍼1 차종4 SP6 *)
    S369_M_이송버퍼1_차종4_SP7 : BOOL; (* AT %MW10322.15 *) (* S369 M 이송버퍼1 차종4 SP7 *)
    S369_M_이송버퍼1_차종4_내수 : BOOL; (* AT %MW10322.0 *) (* S369 M 이송버퍼1 차종4 내수 *)
    S369_M_이송버퍼1_차종4_러시아 : BOOL; (* AT %MW10322.10 *) (* S369 M 이송버퍼1 차종4 러시아 *)
    S369_M_이송버퍼1_차종4_북미 : BOOL; (* AT %MW10322.2 *) (* S369 M 이송버퍼1 차종4 북미 *)
    S369_M_이송버퍼1_차종4_브라질 : BOOL; (* AT %MW10322.7 *) (* S369 M 이송버퍼1 차종4 브라질 *)
    S369_M_이송버퍼1_차종4_수출 : BOOL; (* AT %MW10322.1 *) (* S369 M 이송버퍼1 차종4 수출 *)
    S369_M_이송버퍼1_차종4_중국 : BOOL; (* AT %MW10322.6 *) (* S369 M 이송버퍼1 차종4 중국 *)
    S369_M_이송버퍼1_차종4_중동 : BOOL; (* AT %MW10322.5 *) (* S369 M 이송버퍼1 차종4 중동 *)
    S369_M_이송버퍼1_차종4_호주 : BOOL; (* AT %MW10322.4 *) (* S369 M 이송버퍼1 차종4 호주 *)
    S369_M_이송버퍼1_차종5_AT : BOOL; (* AT %MW10323.1 *) (* S369 M 이송버퍼1 차종5 AT *)
    S369_M_이송버퍼1_차종5_MT : BOOL; (* AT %MW10323.0 *) (* S369 M 이송버퍼1 차종5 MT *)
    S369_M_이송버퍼1_차종5_SP1 : BOOL; (* AT %MW10323.2 *) (* S369 M 이송버퍼1 차종5 SP1 *)
    S369_M_이송버퍼1_차종6_DSROOF : BOOL; (* AT %MW10323.6 *) (* S369 M 이송버퍼1 차종6 DSROOF *)
    S369_M_이송버퍼1_차종6_SP1 : BOOL; (* AT %MW10323.7 *) (* S369 M 이송버퍼1 차종6 SP1 *)
    S369_M_이송버퍼1_차종6_썬루프 : BOOL; (* AT %MW10323.4 *) (* S369 M 이송버퍼1 차종6 썬루프 *)
    S369_M_이송버퍼1_차종6_일반루프 : BOOL; (* AT %MW10323.3 *) (* S369 M 이송버퍼1 차종6 일반루프 *)
    S369_M_이송버퍼1_차종6_파노라마루프 : BOOL; (* AT %MW10323.5 *) (* S369 M 이송버퍼1 차종6 파노라마루프 *)
    S369_M_이송버퍼1_차종7_DSL : BOOL; (* AT %MW10323.9 *) (* S369 M 이송버퍼1 차종7 DSL *)
    S369_M_이송버퍼1_차종7_GSL : BOOL; (* AT %MW10323.8 *) (* S369 M 이송버퍼1 차종7 GSL *)
    S369_M_이송버퍼1_차종7_SP1 : BOOL; (* AT %MW10323.10 *) (* S369 M 이송버퍼1 차종7 SP1 *)
    S369_M_이송버퍼1_차종7_SP2 : BOOL; (* AT %MW10323.11 *) (* S369 M 이송버퍼1 차종7 SP2 *)
    S369_M_이송버퍼1_차종7_SP3 : BOOL; (* AT %MW10323.12 *) (* S369 M 이송버퍼1 차종7 SP3 *)
    S369_M_이송버퍼1_차종7_SP4 : BOOL; (* AT %MW10323.13 *) (* S369 M 이송버퍼1 차종7 SP4 *)
    S369_M_이송버퍼1_차종7_SP5 : BOOL; (* AT %MW10323.14 *) (* S369 M 이송버퍼1 차종7 SP5 *)
    S369_M_이송버퍼1_차종7_SP6 : BOOL; (* AT %MW10323.15 *) (* S369 M 이송버퍼1 차종7 SP6 *)
    S369_M_이송버퍼1_차종8_2WD : BOOL; (* AT %MW10324.0 *) (* S369 M 이송버퍼1 차종8 2WD *)
    S369_M_이송버퍼1_차종8_4WD : BOOL; (* AT %MW10324.1 *) (* S369 M 이송버퍼1 차종8 4WD *)
    S369_M_이송버퍼1_차종8_SP1 : BOOL; (* AT %MW10324.2 *) (* S369 M 이송버퍼1 차종8 SP1 *)
    S369_M_이송버퍼1_차종9_MPI : BOOL; (* AT %MW10324.3 *) (* S369 M 이송버퍼1 차종9 MPI *)
    S369_M_이송버퍼1_차종9_SP1 : BOOL; (* AT %MW10324.5 *) (* S369 M 이송버퍼1 차종9 SP1 *)
    S369_M_이송버퍼1_차종9_SP10 : BOOL; (* AT %MW10324.14 *) (* S369 M 이송버퍼1 차종9 SP10 *)
    S369_M_이송버퍼1_차종9_SP11 : BOOL; (* AT %MW10324.15 *) (* S369 M 이송버퍼1 차종9 SP11 *)
    S369_M_이송버퍼1_차종9_SP2 : BOOL; (* AT %MW10324.6 *) (* S369 M 이송버퍼1 차종9 SP2 *)
    S369_M_이송버퍼1_차종9_SP3 : BOOL; (* AT %MW10324.7 *) (* S369 M 이송버퍼1 차종9 SP3 *)
    S369_M_이송버퍼1_차종9_SP4 : BOOL; (* AT %MW10324.8 *) (* S369 M 이송버퍼1 차종9 SP4 *)
    S369_M_이송버퍼1_차종9_SP5 : BOOL; (* AT %MW10324.9 *) (* S369 M 이송버퍼1 차종9 SP5 *)
    S369_M_이송버퍼1_차종9_SP6 : BOOL; (* AT %MW10324.10 *) (* S369 M 이송버퍼1 차종9 SP6 *)
    S369_M_이송버퍼1_차종9_SP7 : BOOL; (* AT %MW10324.11 *) (* S369 M 이송버퍼1 차종9 SP7 *)
    S369_M_이송버퍼1_차종9_SP8 : BOOL; (* AT %MW10324.12 *) (* S369 M 이송버퍼1 차종9 SP8 *)
    S369_M_이송버퍼1_차종9_SP9 : BOOL; (* AT %MW10324.13 *) (* S369 M 이송버퍼1 차종9 SP9 *)
    S369_M_이송버퍼1_차종9_T_GDI : BOOL; (* AT %MW10324.4 *) (* S369 M 이송버퍼1 차종9 T GDI *)
    S369_M_이송버퍼1_차종_OPT1_R_RACK_무 : BOOL; (* AT %MW10325.3 *) (* S369 M 이송버퍼1 차종 OPT1 R RACK 무 *)
    S369_M_이송버퍼1_차종_OPT1_R_RACK_유 : BOOL; (* AT %MW10325.2 *) (* S369 M 이송버퍼1 차종 OPT1 R RACK 유 *)
    S369_M_이송버퍼1_차종_OPT1_S_REP_EATER_무 : BOOL; (* AT %MW10325.7 *) (* S369 M 이송버퍼1 차종 OPT1 S REP EATER 무 *)
    S369_M_이송버퍼1_차종_OPT1_S_REP_EATER_유 : BOOL; (* AT %MW10325.6 *) (* S369 M 이송버퍼1 차종 OPT1 S REP EATER 유 *)
    S369_M_이송버퍼1_차종_OPT1_VAN_무 : BOOL; (* AT %MW10325.9 *) (* S369 M 이송버퍼1 차종 OPT1 VAN 무 *)
    S369_M_이송버퍼1_차종_OPT1_VAN_유 : BOOL; (* AT %MW10325.8 *) (* S369 M 이송버퍼1 차종 OPT1 VAN 유 *)
    S369_M_이송버퍼1_차종_OPT1_슬라이딩_무 : BOOL; (* AT %MW10325.1 *) (* S369 M 이송버퍼1 차종 OPT1 슬라이딩 무 *)
    S369_M_이송버퍼1_차종_OPT1_슬라이딩_유 : BOOL; (* AT %MW10325.0 *) (* S369 M 이송버퍼1 차종 OPT1 슬라이딩 유 *)
    S369_M_이송버퍼1_차종_OPT1_폴딩_무 : BOOL; (* AT %MW10325.5 *) (* S369 M 이송버퍼1 차종 OPT1 폴딩 무 *)
    S369_M_이송버퍼1_차종_OPT1_폴딩_유 : BOOL; (* AT %MW10325.4 *) (* S369 M 이송버퍼1 차종 OPT1 폴딩 유 *)
    S369_M_이송버퍼1_차종_무 : BOOL; (* AT %MW5002.11 *)
    S369_M_이송버퍼1_차종_유 : BOOL; (* AT %MW5002.10 *)
    S369_M_이송버퍼2_SEQ : WORD; (* AT %MW10300 *) (* S369 M 이송버퍼2 SEQ *)
    S369_M_이송버퍼2_차종1_AX : BOOL; (* AT %MW10301.0 *) (* S369 M 이송버퍼2 차종1 AX *)
    S369_M_이송버퍼2_차종1_B : BOOL; (* AT %MW10301.1 *) (* S369 M 이송버퍼2 차종1 B *)
    S369_M_이송버퍼2_차종1_C : BOOL; (* AT %MW10301.2 *) (* S369 M 이송버퍼2 차종1 C *)
    S369_M_이송버퍼2_차종1_D : BOOL; (* AT %MW10301.3 *) (* S369 M 이송버퍼2 차종1 D *)
    S369_M_이송버퍼2_차종1_E : BOOL; (* AT %MW10301.4 *) (* S369 M 이송버퍼2 차종1 E *)
    S369_M_이송버퍼2_차종1_F : BOOL; (* AT %MW10301.5 *) (* S369 M 이송버퍼2 차종1 F *)
    S369_M_이송버퍼2_차종1_G : BOOL; (* AT %MW10301.6 *) (* S369 M 이송버퍼2 차종1 G *)
    S369_M_이송버퍼2_차종1_H : BOOL; (* AT %MW10301.7 *) (* S369 M 이송버퍼2 차종1 H *)
    S369_M_이송버퍼2_차종2_3DR : BOOL; (* AT %MW10301.8 *) (* S369 M 이송버퍼2 차종2 3DR *)
    S369_M_이송버퍼2_차종2_4DR : BOOL; (* AT %MW10301.9 *) (* S369 M 이송버퍼2 차종2 4DR *)
    S369_M_이송버퍼2_차종2_5DR : BOOL; (* AT %MW10301.10 *) (* S369 M 이송버퍼2 차종2 5DR *)
    S369_M_이송버퍼2_차종2_SP1 : BOOL; (* AT %MW10301.12 *) (* S369 M 이송버퍼2 차종2 SP1 *)
    S369_M_이송버퍼2_차종2_SP2 : BOOL; (* AT %MW10301.13 *) (* S369 M 이송버퍼2 차종2 SP2 *)
    S369_M_이송버퍼2_차종2_WGN : BOOL; (* AT %MW10301.11 *) (* S369 M 이송버퍼2 차종2 WGN *)
    S369_M_이송버퍼2_차종3_LHD : BOOL; (* AT %MW10301.14 *) (* S369 M 이송버퍼2 차종3 LHD *)
    S369_M_이송버퍼2_차종3_RHD : BOOL; (* AT %MW10301.15 *) (* S369 M 이송버퍼2 차종3 RHD *)
    S369_M_이송버퍼2_차종4_EEC : BOOL; (* AT %MW10302.3 *) (* S369 M 이송버퍼2 차종4 EEC *)
    S369_M_이송버퍼2_차종4_SP1 : BOOL; (* AT %MW10302.8 *) (* S369 M 이송버퍼2 차종4 SP1 *)
    S369_M_이송버퍼2_차종4_SP2 : BOOL; (* AT %MW10302.9 *) (* S369 M 이송버퍼2 차종4 SP2 *)
    S369_M_이송버퍼2_차종4_SP3 : BOOL; (* AT %MW10302.11 *) (* S369 M 이송버퍼2 차종4 SP3 *)
    S369_M_이송버퍼2_차종4_SP4 : BOOL; (* AT %MW10302.12 *) (* S369 M 이송버퍼2 차종4 SP4 *)
    S369_M_이송버퍼2_차종4_SP5 : BOOL; (* AT %MW10302.13 *) (* S369 M 이송버퍼2 차종4 SP5 *)
    S369_M_이송버퍼2_차종4_SP6 : BOOL; (* AT %MW10302.14 *) (* S369 M 이송버퍼2 차종4 SP6 *)
    S369_M_이송버퍼2_차종4_SP7 : BOOL; (* AT %MW10302.15 *) (* S369 M 이송버퍼2 차종4 SP7 *)
    S369_M_이송버퍼2_차종4_내수 : BOOL; (* AT %MW10302.0 *) (* S369 M 이송버퍼2 차종4 내수 *)
    S369_M_이송버퍼2_차종4_러시아 : BOOL; (* AT %MW10302.10 *) (* S369 M 이송버퍼2 차종4 러시아 *)
    S369_M_이송버퍼2_차종4_북미 : BOOL; (* AT %MW10302.2 *) (* S369 M 이송버퍼2 차종4 북미 *)
    S369_M_이송버퍼2_차종4_브라질 : BOOL; (* AT %MW10302.7 *) (* S369 M 이송버퍼2 차종4 브라질 *)
    S369_M_이송버퍼2_차종4_수출 : BOOL; (* AT %MW10302.1 *) (* S369 M 이송버퍼2 차종4 수출 *)
    S369_M_이송버퍼2_차종4_중국 : BOOL; (* AT %MW10302.6 *) (* S369 M 이송버퍼2 차종4 중국 *)
    S369_M_이송버퍼2_차종4_중동 : BOOL; (* AT %MW10302.5 *) (* S369 M 이송버퍼2 차종4 중동 *)
    S369_M_이송버퍼2_차종4_호주 : BOOL; (* AT %MW10302.4 *) (* S369 M 이송버퍼2 차종4 호주 *)
    S369_M_이송버퍼2_차종5_AT : BOOL; (* AT %MW10303.1 *) (* S369 M 이송버퍼2 차종5 AT *)
    S369_M_이송버퍼2_차종5_MT : BOOL; (* AT %MW10303.0 *) (* S369 M 이송버퍼2 차종5 MT *)
    S369_M_이송버퍼2_차종5_SP1 : BOOL; (* AT %MW10303.2 *) (* S369 M 이송버퍼2 차종5 SP1 *)
    S369_M_이송버퍼2_차종6_DSROOF : BOOL; (* AT %MW10303.6 *) (* S369 M 이송버퍼2 차종6 DSROOF *)
    S369_M_이송버퍼2_차종6_SP1 : BOOL; (* AT %MW10303.7 *) (* S369 M 이송버퍼2 차종6 SP1 *)
    S369_M_이송버퍼2_차종6_썬루프 : BOOL; (* AT %MW10303.4 *) (* S369 M 이송버퍼2 차종6 썬루프 *)
    S369_M_이송버퍼2_차종6_일반루프 : BOOL; (* AT %MW10303.3 *) (* S369 M 이송버퍼2 차종6 일반루프 *)
    S369_M_이송버퍼2_차종6_파노라마루프 : BOOL; (* AT %MW10303.5 *) (* S369 M 이송버퍼2 차종6 파노라마루프 *)
    S369_M_이송버퍼2_차종7_DSL : BOOL; (* AT %MW10303.9 *) (* S369 M 이송버퍼2 차종7 DSL *)
    S369_M_이송버퍼2_차종7_GSL : BOOL; (* AT %MW10303.8 *) (* S369 M 이송버퍼2 차종7 GSL *)
    S369_M_이송버퍼2_차종7_SP1 : BOOL; (* AT %MW10303.10 *) (* S369 M 이송버퍼2 차종7 SP1 *)
    S369_M_이송버퍼2_차종7_SP2 : BOOL; (* AT %MW10303.11 *) (* S369 M 이송버퍼2 차종7 SP2 *)
    S369_M_이송버퍼2_차종7_SP3 : BOOL; (* AT %MW10303.12 *) (* S369 M 이송버퍼2 차종7 SP3 *)
    S369_M_이송버퍼2_차종7_SP4 : BOOL; (* AT %MW10303.13 *) (* S369 M 이송버퍼2 차종7 SP4 *)
    S369_M_이송버퍼2_차종7_SP5 : BOOL; (* AT %MW10303.14 *) (* S369 M 이송버퍼2 차종7 SP5 *)
    S369_M_이송버퍼2_차종7_SP6 : BOOL; (* AT %MW10303.15 *) (* S369 M 이송버퍼2 차종7 SP6 *)
    S369_M_이송버퍼2_차종8_2WD : BOOL; (* AT %MW10304.0 *) (* S369 M 이송버퍼2 차종8 2WD *)
    S369_M_이송버퍼2_차종8_4WD : BOOL; (* AT %MW10304.1 *) (* S369 M 이송버퍼2 차종8 4WD *)
    S369_M_이송버퍼2_차종8_SP1 : BOOL; (* AT %MW10304.2 *) (* S369 M 이송버퍼2 차종8 SP1 *)
    S369_M_이송버퍼2_차종9_MPI : BOOL; (* AT %MW10304.3 *) (* S369 M 이송버퍼2 차종9 MPI *)
    S369_M_이송버퍼2_차종9_SP1 : BOOL; (* AT %MW10304.5 *) (* S369 M 이송버퍼2 차종9 SP1 *)
    S369_M_이송버퍼2_차종9_SP10 : BOOL; (* AT %MW10304.14 *) (* S369 M 이송버퍼2 차종9 SP10 *)
    S369_M_이송버퍼2_차종9_SP11 : BOOL; (* AT %MW10304.15 *) (* S369 M 이송버퍼2 차종9 SP11 *)
    S369_M_이송버퍼2_차종9_SP2 : BOOL; (* AT %MW10304.6 *) (* S369 M 이송버퍼2 차종9 SP2 *)
    S369_M_이송버퍼2_차종9_SP3 : BOOL; (* AT %MW10304.7 *) (* S369 M 이송버퍼2 차종9 SP3 *)
    S369_M_이송버퍼2_차종9_SP4 : BOOL; (* AT %MW10304.8 *) (* S369 M 이송버퍼2 차종9 SP4 *)
    S369_M_이송버퍼2_차종9_SP5 : BOOL; (* AT %MW10304.9 *) (* S369 M 이송버퍼2 차종9 SP5 *)
    S369_M_이송버퍼2_차종9_SP6 : BOOL; (* AT %MW10304.10 *) (* S369 M 이송버퍼2 차종9 SP6 *)
    S369_M_이송버퍼2_차종9_SP7 : BOOL; (* AT %MW10304.11 *) (* S369 M 이송버퍼2 차종9 SP7 *)
    S369_M_이송버퍼2_차종9_SP8 : BOOL; (* AT %MW10304.12 *) (* S369 M 이송버퍼2 차종9 SP8 *)
    S369_M_이송버퍼2_차종9_SP9 : BOOL; (* AT %MW10304.13 *) (* S369 M 이송버퍼2 차종9 SP9 *)
    S369_M_이송버퍼2_차종9_T_GDI : BOOL; (* AT %MW10304.4 *) (* S369 M 이송버퍼2 차종9 T GDI *)
    S369_M_이송버퍼2_차종_OPT1_R_RACK_무 : BOOL; (* AT %MW10305.3 *) (* S369 M 이송버퍼2 차종 OPT1 R RACK 무 *)
    S369_M_이송버퍼2_차종_OPT1_R_RACK_유 : BOOL; (* AT %MW10305.2 *) (* S369 M 이송버퍼2 차종 OPT1 R RACK 유 *)
    S369_M_이송버퍼2_차종_OPT1_S_REP_EATER_무 : BOOL; (* AT %MW10305.7 *) (* S369 M 이송버퍼2 차종 OPT1 S REP EATER 무 *)
    S369_M_이송버퍼2_차종_OPT1_S_REP_EATER_유 : BOOL; (* AT %MW10305.6 *) (* S369 M 이송버퍼2 차종 OPT1 S REP EATER 유 *)
    S369_M_이송버퍼2_차종_OPT1_VAN_무 : BOOL; (* AT %MW10305.9 *) (* S369 M 이송버퍼2 차종 OPT1 VAN 무 *)
    S369_M_이송버퍼2_차종_OPT1_VAN_유 : BOOL; (* AT %MW10305.8 *) (* S369 M 이송버퍼2 차종 OPT1 VAN 유 *)
    S369_M_이송버퍼2_차종_OPT1_슬라이딩_무 : BOOL; (* AT %MW10305.1 *) (* S369 M 이송버퍼2 차종 OPT1 슬라이딩 무 *)
    S369_M_이송버퍼2_차종_OPT1_슬라이딩_유 : BOOL; (* AT %MW10305.0 *) (* S369 M 이송버퍼2 차종 OPT1 슬라이딩 유 *)
    S369_M_이송버퍼2_차종_OPT1_폴딩_무 : BOOL; (* AT %MW10305.5 *) (* S369 M 이송버퍼2 차종 OPT1 폴딩 무 *)
    S369_M_이송버퍼2_차종_OPT1_폴딩_유 : BOOL; (* AT %MW10305.4 *) (* S369 M 이송버퍼2 차종 OPT1 폴딩 유 *)
    S369_M_이송버퍼2_차종_무 : BOOL; (* AT %MW5002.9 *)
    S369_M_이송버퍼2_차종_유 : BOOL; (* AT %MW5002.8 *)
    S369_M_이송버퍼3_SEQ : WORD; (* AT %MW10280 *) (* S369 M 이송버퍼3 SEQ *)
    S369_M_이송버퍼3_차종1_AX : BOOL; (* AT %MW10281.0 *) (* S369 M 이송버퍼3 차종1 AX *)
    S369_M_이송버퍼3_차종1_B : BOOL; (* AT %MW10281.1 *) (* S369 M 이송버퍼3 차종1 B *)
    S369_M_이송버퍼3_차종1_C : BOOL; (* AT %MW10281.2 *) (* S369 M 이송버퍼3 차종1 C *)
    S369_M_이송버퍼3_차종1_D : BOOL; (* AT %MW10281.3 *) (* S369 M 이송버퍼3 차종1 D *)
    S369_M_이송버퍼3_차종1_E : BOOL; (* AT %MW10281.4 *) (* S369 M 이송버퍼3 차종1 E *)
    S369_M_이송버퍼3_차종1_F : BOOL; (* AT %MW10281.5 *) (* S369 M 이송버퍼3 차종1 F *)
    S369_M_이송버퍼3_차종1_G : BOOL; (* AT %MW10281.6 *) (* S369 M 이송버퍼3 차종1 G *)
    S369_M_이송버퍼3_차종1_H : BOOL; (* AT %MW10281.7 *) (* S369 M 이송버퍼3 차종1 H *)
    S369_M_이송버퍼3_차종2_3DR : BOOL; (* AT %MW10281.8 *) (* S369 M 이송버퍼3 차종2 3DR *)
    S369_M_이송버퍼3_차종2_4DR : BOOL; (* AT %MW10281.9 *) (* S369 M 이송버퍼3 차종2 4DR *)
    S369_M_이송버퍼3_차종2_5DR : BOOL; (* AT %MW10281.10 *) (* S369 M 이송버퍼3 차종2 5DR *)
    S369_M_이송버퍼3_차종2_SP1 : BOOL; (* AT %MW10281.12 *) (* S369 M 이송버퍼3 차종2 SP1 *)
    S369_M_이송버퍼3_차종2_SP2 : BOOL; (* AT %MW10281.13 *) (* S369 M 이송버퍼3 차종2 SP2 *)
    S369_M_이송버퍼3_차종2_WGN : BOOL; (* AT %MW10281.11 *) (* S369 M 이송버퍼3 차종2 WGN *)
    S369_M_이송버퍼3_차종3_LHD : BOOL; (* AT %MW10281.14 *) (* S369 M 이송버퍼3 차종3 LHD *)
    S369_M_이송버퍼3_차종3_RHD : BOOL; (* AT %MW10281.15 *) (* S369 M 이송버퍼3 차종3 RHD *)
    S369_M_이송버퍼3_차종4_EEC : BOOL; (* AT %MW10282.3 *) (* S369 M 이송버퍼3 차종4 EEC *)
    S369_M_이송버퍼3_차종4_SP1 : BOOL; (* AT %MW10282.8 *) (* S369 M 이송버퍼3 차종4 SP1 *)
    S369_M_이송버퍼3_차종4_SP2 : BOOL; (* AT %MW10282.9 *) (* S369 M 이송버퍼3 차종4 SP2 *)
    S369_M_이송버퍼3_차종4_SP3 : BOOL; (* AT %MW10282.11 *) (* S369 M 이송버퍼3 차종4 SP3 *)
    S369_M_이송버퍼3_차종4_SP4 : BOOL; (* AT %MW10282.12 *) (* S369 M 이송버퍼3 차종4 SP4 *)
    S369_M_이송버퍼3_차종4_SP5 : BOOL; (* AT %MW10282.13 *) (* S369 M 이송버퍼3 차종4 SP5 *)
    S369_M_이송버퍼3_차종4_SP6 : BOOL; (* AT %MW10282.14 *) (* S369 M 이송버퍼3 차종4 SP6 *)
    S369_M_이송버퍼3_차종4_SP7 : BOOL; (* AT %MW10282.15 *) (* S369 M 이송버퍼3 차종4 SP7 *)
    S369_M_이송버퍼3_차종4_내수 : BOOL; (* AT %MW10282.0 *) (* S369 M 이송버퍼3 차종4 내수 *)
    S369_M_이송버퍼3_차종4_러시아 : BOOL; (* AT %MW10282.10 *) (* S369 M 이송버퍼3 차종4 러시아 *)
    S369_M_이송버퍼3_차종4_북미 : BOOL; (* AT %MW10282.2 *) (* S369 M 이송버퍼3 차종4 북미 *)
    S369_M_이송버퍼3_차종4_브라질 : BOOL; (* AT %MW10282.7 *) (* S369 M 이송버퍼3 차종4 브라질 *)
    S369_M_이송버퍼3_차종4_수출 : BOOL; (* AT %MW10282.1 *) (* S369 M 이송버퍼3 차종4 수출 *)
    S369_M_이송버퍼3_차종4_중국 : BOOL; (* AT %MW10282.6 *) (* S369 M 이송버퍼3 차종4 중국 *)
    S369_M_이송버퍼3_차종4_중동 : BOOL; (* AT %MW10282.5 *) (* S369 M 이송버퍼3 차종4 중동 *)
    S369_M_이송버퍼3_차종4_호주 : BOOL; (* AT %MW10282.4 *) (* S369 M 이송버퍼3 차종4 호주 *)
    S369_M_이송버퍼3_차종5_AT : BOOL; (* AT %MW10283.1 *) (* S369 M 이송버퍼3 차종5 AT *)
    S369_M_이송버퍼3_차종5_MT : BOOL; (* AT %MW10283.0 *) (* S369 M 이송버퍼3 차종5 MT *)
    S369_M_이송버퍼3_차종5_SP1 : BOOL; (* AT %MW10283.2 *) (* S369 M 이송버퍼3 차종5 SP1 *)
    S369_M_이송버퍼3_차종6_DSROOF : BOOL; (* AT %MW10283.6 *) (* S369 M 이송버퍼3 차종6 DSROOF *)
    S369_M_이송버퍼3_차종6_SP1 : BOOL; (* AT %MW10283.7 *) (* S369 M 이송버퍼3 차종6 SP1 *)
    S369_M_이송버퍼3_차종6_썬루프 : BOOL; (* AT %MW10283.4 *) (* S369 M 이송버퍼3 차종6 썬루프 *)
    S369_M_이송버퍼3_차종6_일반루프 : BOOL; (* AT %MW10283.3 *) (* S369 M 이송버퍼3 차종6 일반루프 *)
    S369_M_이송버퍼3_차종6_파노라마루프 : BOOL; (* AT %MW10283.5 *) (* S369 M 이송버퍼3 차종6 파노라마루프 *)
    S369_M_이송버퍼3_차종7_DSL : BOOL; (* AT %MW10283.9 *) (* S369 M 이송버퍼3 차종7 DSL *)
    S369_M_이송버퍼3_차종7_GSL : BOOL; (* AT %MW10283.8 *) (* S369 M 이송버퍼3 차종7 GSL *)
    S369_M_이송버퍼3_차종7_SP1 : BOOL; (* AT %MW10283.10 *) (* S369 M 이송버퍼3 차종7 SP1 *)
    S369_M_이송버퍼3_차종7_SP2 : BOOL; (* AT %MW10283.11 *) (* S369 M 이송버퍼3 차종7 SP2 *)
    S369_M_이송버퍼3_차종7_SP3 : BOOL; (* AT %MW10283.12 *) (* S369 M 이송버퍼3 차종7 SP3 *)
    S369_M_이송버퍼3_차종7_SP4 : BOOL; (* AT %MW10283.13 *) (* S369 M 이송버퍼3 차종7 SP4 *)
    S369_M_이송버퍼3_차종7_SP5 : BOOL; (* AT %MW10283.14 *) (* S369 M 이송버퍼3 차종7 SP5 *)
    S369_M_이송버퍼3_차종7_SP6 : BOOL; (* AT %MW10283.15 *) (* S369 M 이송버퍼3 차종7 SP6 *)
    S369_M_이송버퍼3_차종8_2WD : BOOL; (* AT %MW10284.0 *) (* S369 M 이송버퍼3 차종8 2WD *)
    S369_M_이송버퍼3_차종8_4WD : BOOL; (* AT %MW10284.1 *) (* S369 M 이송버퍼3 차종8 4WD *)
    S369_M_이송버퍼3_차종8_SP1 : BOOL; (* AT %MW10284.2 *) (* S369 M 이송버퍼3 차종8 SP1 *)
    S369_M_이송버퍼3_차종9_MPI : BOOL; (* AT %MW10284.3 *) (* S369 M 이송버퍼3 차종9 MPI *)
    S369_M_이송버퍼3_차종9_SP1 : BOOL; (* AT %MW10284.5 *) (* S369 M 이송버퍼3 차종9 SP1 *)
    S369_M_이송버퍼3_차종9_SP10 : BOOL; (* AT %MW10284.14 *) (* S369 M 이송버퍼3 차종9 SP10 *)
    S369_M_이송버퍼3_차종9_SP11 : BOOL; (* AT %MW10284.15 *) (* S369 M 이송버퍼3 차종9 SP11 *)
    S369_M_이송버퍼3_차종9_SP2 : BOOL; (* AT %MW10284.6 *) (* S369 M 이송버퍼3 차종9 SP2 *)
    S369_M_이송버퍼3_차종9_SP3 : BOOL; (* AT %MW10284.7 *) (* S369 M 이송버퍼3 차종9 SP3 *)
    S369_M_이송버퍼3_차종9_SP4 : BOOL; (* AT %MW10284.8 *) (* S369 M 이송버퍼3 차종9 SP4 *)
    S369_M_이송버퍼3_차종9_SP5 : BOOL; (* AT %MW10284.9 *) (* S369 M 이송버퍼3 차종9 SP5 *)
    S369_M_이송버퍼3_차종9_SP6 : BOOL; (* AT %MW10284.10 *) (* S369 M 이송버퍼3 차종9 SP6 *)
    S369_M_이송버퍼3_차종9_SP7 : BOOL; (* AT %MW10284.11 *) (* S369 M 이송버퍼3 차종9 SP7 *)
    S369_M_이송버퍼3_차종9_SP8 : BOOL; (* AT %MW10284.12 *) (* S369 M 이송버퍼3 차종9 SP8 *)
    S369_M_이송버퍼3_차종9_SP9 : BOOL; (* AT %MW10284.13 *) (* S369 M 이송버퍼3 차종9 SP9 *)
    S369_M_이송버퍼3_차종9_T_GDI : BOOL; (* AT %MW10284.4 *) (* S369 M 이송버퍼3 차종9 T GDI *)
    S369_M_이송버퍼3_차종_OPT1_R_RACK_무 : BOOL; (* AT %MW10285.3 *) (* S369 M 이송버퍼3 차종 OPT1 R RACK 무 *)
    S369_M_이송버퍼3_차종_OPT1_R_RACK_유 : BOOL; (* AT %MW10285.2 *) (* S369 M 이송버퍼3 차종 OPT1 R RACK 유 *)
    S369_M_이송버퍼3_차종_OPT1_S_REP_EATER_무 : BOOL; (* AT %MW10285.7 *) (* S369 M 이송버퍼3 차종 OPT1 S REP EATER 무 *)
    S369_M_이송버퍼3_차종_OPT1_S_REP_EATER_유 : BOOL; (* AT %MW10285.6 *) (* S369 M 이송버퍼3 차종 OPT1 S REP EATER 유 *)
    S369_M_이송버퍼3_차종_OPT1_VAN_무 : BOOL; (* AT %MW10285.9 *) (* S369 M 이송버퍼3 차종 OPT1 VAN 무 *)
    S369_M_이송버퍼3_차종_OPT1_VAN_유 : BOOL; (* AT %MW10285.8 *) (* S369 M 이송버퍼3 차종 OPT1 VAN 유 *)
    S369_M_이송버퍼3_차종_OPT1_슬라이딩_무 : BOOL; (* AT %MW10285.1 *) (* S369 M 이송버퍼3 차종 OPT1 슬라이딩 무 *)
    S369_M_이송버퍼3_차종_OPT1_슬라이딩_유 : BOOL; (* AT %MW10285.0 *) (* S369 M 이송버퍼3 차종 OPT1 슬라이딩 유 *)
    S369_M_이송버퍼3_차종_OPT1_폴딩_무 : BOOL; (* AT %MW10285.5 *) (* S369 M 이송버퍼3 차종 OPT1 폴딩 무 *)
    S369_M_이송버퍼3_차종_OPT1_폴딩_유 : BOOL; (* AT %MW10285.4 *) (* S369 M 이송버퍼3 차종 OPT1 폴딩 유 *)
    S369_M_이송버퍼3_차종_무 : BOOL; (* AT %MW5002.7 *)
    S369_M_이송버퍼3_차종_유 : BOOL; (* AT %MW5002.6 *)
    S369_M_이송버퍼4_SEQ : WORD; (* AT %MW10260 *) (* S369 M 이송버퍼4 SEQ *)
    S369_M_이송버퍼4_도착완료 : BOOL; (* AT %MW5003.2 *)
    S369_M_이송버퍼4_차종1_AX : BOOL; (* AT %MW10261.0 *) (* S369 M 이송버퍼4 차종1 AX *)
    S369_M_이송버퍼4_차종1_B : BOOL; (* AT %MW10261.1 *) (* S369 M 이송버퍼4 차종1 B *)
    S369_M_이송버퍼4_차종1_C : BOOL; (* AT %MW10261.2 *) (* S369 M 이송버퍼4 차종1 C *)
    S369_M_이송버퍼4_차종1_D : BOOL; (* AT %MW10261.3 *) (* S369 M 이송버퍼4 차종1 D *)
    S369_M_이송버퍼4_차종1_E : BOOL; (* AT %MW10261.4 *) (* S369 M 이송버퍼4 차종1 E *)
    S369_M_이송버퍼4_차종1_F : BOOL; (* AT %MW10261.5 *) (* S369 M 이송버퍼4 차종1 F *)
    S369_M_이송버퍼4_차종1_G : BOOL; (* AT %MW10261.6 *) (* S369 M 이송버퍼4 차종1 G *)
    S369_M_이송버퍼4_차종1_H : BOOL; (* AT %MW10261.7 *) (* S369 M 이송버퍼4 차종1 H *)
    S369_M_이송버퍼4_차종2_3DR : BOOL; (* AT %MW10261.8 *) (* S369 M 이송버퍼4 차종2 3DR *)
    S369_M_이송버퍼4_차종2_4DR : BOOL; (* AT %MW10261.9 *) (* S369 M 이송버퍼4 차종2 4DR *)
    S369_M_이송버퍼4_차종2_5DR : BOOL; (* AT %MW10261.10 *) (* S369 M 이송버퍼4 차종2 5DR *)
    S369_M_이송버퍼4_차종2_SP1 : BOOL; (* AT %MW10261.12 *) (* S369 M 이송버퍼4 차종2 SP1 *)
    S369_M_이송버퍼4_차종2_SP2 : BOOL; (* AT %MW10261.13 *) (* S369 M 이송버퍼4 차종2 SP2 *)
    S369_M_이송버퍼4_차종2_WGN : BOOL; (* AT %MW10261.11 *) (* S369 M 이송버퍼4 차종2 WGN *)
    S369_M_이송버퍼4_차종3_LHD : BOOL; (* AT %MW10261.14 *) (* S369 M 이송버퍼4 차종3 LHD *)
    S369_M_이송버퍼4_차종3_RHD : BOOL; (* AT %MW10261.15 *) (* S369 M 이송버퍼4 차종3 RHD *)
    S369_M_이송버퍼4_차종4_EEC : BOOL; (* AT %MW10262.3 *) (* S369 M 이송버퍼4 차종4 EEC *)
    S369_M_이송버퍼4_차종4_SP1 : BOOL; (* AT %MW10262.8 *) (* S369 M 이송버퍼4 차종4 SP1 *)
    S369_M_이송버퍼4_차종4_SP2 : BOOL; (* AT %MW10262.9 *) (* S369 M 이송버퍼4 차종4 SP2 *)
    S369_M_이송버퍼4_차종4_SP3 : BOOL; (* AT %MW10262.11 *) (* S369 M 이송버퍼4 차종4 SP3 *)
    S369_M_이송버퍼4_차종4_SP4 : BOOL; (* AT %MW10262.12 *) (* S369 M 이송버퍼4 차종4 SP4 *)
    S369_M_이송버퍼4_차종4_SP5 : BOOL; (* AT %MW10262.13 *) (* S369 M 이송버퍼4 차종4 SP5 *)
    S369_M_이송버퍼4_차종4_SP6 : BOOL; (* AT %MW10262.14 *) (* S369 M 이송버퍼4 차종4 SP6 *)
    S369_M_이송버퍼4_차종4_SP7 : BOOL; (* AT %MW10262.15 *) (* S369 M 이송버퍼4 차종4 SP7 *)
    S369_M_이송버퍼4_차종4_내수 : BOOL; (* AT %MW10262.0 *) (* S369 M 이송버퍼4 차종4 내수 *)
    S369_M_이송버퍼4_차종4_러시아 : BOOL; (* AT %MW10262.10 *) (* S369 M 이송버퍼4 차종4 러시아 *)
    S369_M_이송버퍼4_차종4_북미 : BOOL; (* AT %MW10262.2 *) (* S369 M 이송버퍼4 차종4 북미 *)
    S369_M_이송버퍼4_차종4_브라질 : BOOL; (* AT %MW10262.7 *) (* S369 M 이송버퍼4 차종4 브라질 *)
    S369_M_이송버퍼4_차종4_수출 : BOOL; (* AT %MW10262.1 *) (* S369 M 이송버퍼4 차종4 수출 *)
    S369_M_이송버퍼4_차종4_중국 : BOOL; (* AT %MW10262.6 *) (* S369 M 이송버퍼4 차종4 중국 *)
    S369_M_이송버퍼4_차종4_중동 : BOOL; (* AT %MW10262.5 *) (* S369 M 이송버퍼4 차종4 중동 *)
    S369_M_이송버퍼4_차종4_호주 : BOOL; (* AT %MW10262.4 *) (* S369 M 이송버퍼4 차종4 호주 *)
    S369_M_이송버퍼4_차종5_AT : BOOL; (* AT %MW10263.1 *) (* S369 M 이송버퍼4 차종5 AT *)
    S369_M_이송버퍼4_차종5_MT : BOOL; (* AT %MW10263.0 *) (* S369 M 이송버퍼4 차종5 MT *)
    S369_M_이송버퍼4_차종5_SP1 : BOOL; (* AT %MW10263.2 *) (* S369 M 이송버퍼4 차종5 SP1 *)
    S369_M_이송버퍼4_차종6_DSROOF : BOOL; (* AT %MW10263.6 *) (* S369 M 이송버퍼4 차종6 DSROOF *)
    S369_M_이송버퍼4_차종6_SP1 : BOOL; (* AT %MW10263.7 *) (* S369 M 이송버퍼4 차종6 SP1 *)
    S369_M_이송버퍼4_차종6_썬루프 : BOOL; (* AT %MW10263.4 *) (* S369 M 이송버퍼4 차종6 썬루프 *)
    S369_M_이송버퍼4_차종6_일반루프 : BOOL; (* AT %MW10263.3 *) (* S369 M 이송버퍼4 차종6 일반루프 *)
    S369_M_이송버퍼4_차종6_파노라마루프 : BOOL; (* AT %MW10263.5 *) (* S369 M 이송버퍼4 차종6 파노라마루프 *)
    S369_M_이송버퍼4_차종7_DSL : BOOL; (* AT %MW10263.9 *) (* S369 M 이송버퍼4 차종7 DSL *)
    S369_M_이송버퍼4_차종7_GSL : BOOL; (* AT %MW10263.8 *) (* S369 M 이송버퍼4 차종7 GSL *)
    S369_M_이송버퍼4_차종7_SP1 : BOOL; (* AT %MW10263.10 *) (* S369 M 이송버퍼4 차종7 SP1 *)
    S369_M_이송버퍼4_차종7_SP2 : BOOL; (* AT %MW10263.11 *) (* S369 M 이송버퍼4 차종7 SP2 *)
    S369_M_이송버퍼4_차종7_SP3 : BOOL; (* AT %MW10263.12 *) (* S369 M 이송버퍼4 차종7 SP3 *)
    S369_M_이송버퍼4_차종7_SP4 : BOOL; (* AT %MW10263.13 *) (* S369 M 이송버퍼4 차종7 SP4 *)
    S369_M_이송버퍼4_차종7_SP5 : BOOL; (* AT %MW10263.14 *) (* S369 M 이송버퍼4 차종7 SP5 *)
    S369_M_이송버퍼4_차종7_SP6 : BOOL; (* AT %MW10263.15 *) (* S369 M 이송버퍼4 차종7 SP6 *)
    S369_M_이송버퍼4_차종8_2WD : BOOL; (* AT %MW10264.0 *) (* S369 M 이송버퍼4 차종8 2WD *)
    S369_M_이송버퍼4_차종8_4WD : BOOL; (* AT %MW10264.1 *) (* S369 M 이송버퍼4 차종8 4WD *)
    S369_M_이송버퍼4_차종8_SP1 : BOOL; (* AT %MW10264.2 *) (* S369 M 이송버퍼4 차종8 SP1 *)
    S369_M_이송버퍼4_차종9_MPI : BOOL; (* AT %MW10264.3 *) (* S369 M 이송버퍼4 차종9 MPI *)
    S369_M_이송버퍼4_차종9_SP1 : BOOL; (* AT %MW10264.5 *) (* S369 M 이송버퍼4 차종9 SP1 *)
    S369_M_이송버퍼4_차종9_SP10 : BOOL; (* AT %MW10264.14 *) (* S369 M 이송버퍼4 차종9 SP10 *)
    S369_M_이송버퍼4_차종9_SP11 : BOOL; (* AT %MW10264.15 *) (* S369 M 이송버퍼4 차종9 SP11 *)
    S369_M_이송버퍼4_차종9_SP2 : BOOL; (* AT %MW10264.6 *) (* S369 M 이송버퍼4 차종9 SP2 *)
    S369_M_이송버퍼4_차종9_SP3 : BOOL; (* AT %MW10264.7 *) (* S369 M 이송버퍼4 차종9 SP3 *)
    S369_M_이송버퍼4_차종9_SP4 : BOOL; (* AT %MW10264.8 *) (* S369 M 이송버퍼4 차종9 SP4 *)
    S369_M_이송버퍼4_차종9_SP5 : BOOL; (* AT %MW10264.9 *) (* S369 M 이송버퍼4 차종9 SP5 *)
    S369_M_이송버퍼4_차종9_SP6 : BOOL; (* AT %MW10264.10 *) (* S369 M 이송버퍼4 차종9 SP6 *)
    S369_M_이송버퍼4_차종9_SP7 : BOOL; (* AT %MW10264.11 *) (* S369 M 이송버퍼4 차종9 SP7 *)
    S369_M_이송버퍼4_차종9_SP8 : BOOL; (* AT %MW10264.12 *) (* S369 M 이송버퍼4 차종9 SP8 *)
    S369_M_이송버퍼4_차종9_SP9 : BOOL; (* AT %MW10264.13 *) (* S369 M 이송버퍼4 차종9 SP9 *)
    S369_M_이송버퍼4_차종9_T_GDI : BOOL; (* AT %MW10264.4 *) (* S369 M 이송버퍼4 차종9 T GDI *)
    S369_M_이송버퍼4_차종_OPT1_R_RACK_무 : BOOL; (* AT %MW10265.3 *) (* S369 M 이송버퍼4 차종 OPT1 R RACK 무 *)
    S369_M_이송버퍼4_차종_OPT1_R_RACK_유 : BOOL; (* AT %MW10265.2 *) (* S369 M 이송버퍼4 차종 OPT1 R RACK 유 *)
    S369_M_이송버퍼4_차종_OPT1_S_REP_EATER_무 : BOOL; (* AT %MW10265.7 *) (* S369 M 이송버퍼4 차종 OPT1 S REP EATER 무 *)
    S369_M_이송버퍼4_차종_OPT1_S_REP_EATER_유 : BOOL; (* AT %MW10265.6 *) (* S369 M 이송버퍼4 차종 OPT1 S REP EATER 유 *)
    S369_M_이송버퍼4_차종_OPT1_VAN_무 : BOOL; (* AT %MW10265.9 *) (* S369 M 이송버퍼4 차종 OPT1 VAN 무 *)
    S369_M_이송버퍼4_차종_OPT1_VAN_유 : BOOL; (* AT %MW10265.8 *) (* S369 M 이송버퍼4 차종 OPT1 VAN 유 *)
    S369_M_이송버퍼4_차종_OPT1_슬라이딩_무 : BOOL; (* AT %MW10265.1 *) (* S369 M 이송버퍼4 차종 OPT1 슬라이딩 무 *)
    S369_M_이송버퍼4_차종_OPT1_슬라이딩_유 : BOOL; (* AT %MW10265.0 *) (* S369 M 이송버퍼4 차종 OPT1 슬라이딩 유 *)
    S369_M_이송버퍼4_차종_OPT1_폴딩_무 : BOOL; (* AT %MW10265.5 *) (* S369 M 이송버퍼4 차종 OPT1 폴딩 무 *)
    S369_M_이송버퍼4_차종_OPT1_폴딩_유 : BOOL; (* AT %MW10265.4 *) (* S369 M 이송버퍼4 차종 OPT1 폴딩 유 *)
    S369_M_이송버퍼4_차종_무 : BOOL; (* AT %MW5002.5 *)
    S369_M_이송버퍼4_차종_유 : BOOL; (* AT %MW5002.4 *)
    S369_M_자동_START : BOOL; (* AT %MW5000.5 *) (* S369 자동운전중 *)
    S369_M_자동_운전중 : BOOL; (* AT %MW5000.4 *) (* S369 자동운전중 *)
    S369_M_자동모드 : BOOL; (* AT %MW5000.1 *) (* S369 선택 자동모드 *)
    S369_M_총괄_이상 : BOOL; (* AT %MW5009.0 *) (* S369_M_총괄_이상 *)
    전체_M_GATE_자동기동 : BOOL; (* AT %MW308.1 *) (* 전체_M_자동_운전 *)
    전체_라인_M_총괄_SAFETY_이상 : BOOL; (* AT %MW300.2 *) (* ALL공정 SAFETY  이상총괄 *)
    전체_라인_M_총괄_공기압_이상 : BOOL; (* AT %MW300.3 *) (* ALL공정 공기압 이상총괄 *)
    전체_라인_M_총괄_비상정지_이상 : BOOL; (* AT %MW300.1 *) (* ALL공정 비상정지 이상총괄 *)
    전체_라인_M_총괄_이상 : BOOL; (* AT %MW300.0 *) (* ALL공정 총괄이상 *)
END_VAR
VAR_EXTERNAL
    BB_MAIN_I_1차_작업완료 : BOOL; (* AT %MW83011.5 *)
    BB_MAIN_I_2차_작업완료 : BOOL; (* AT %MW83011.6 *)
    BB_MAIN_I_불간섭 : BOOL; (* AT %MW83011.0 *)
    BB_MAIN_I_취출완료 : BOOL; (* AT %MW83011.9 *)
    BB_MAIN_I_행거클램프_완료 : BOOL; (* AT %MW83011.8 *)
    EGIS_CWS : BOOL;
    HOP_PBL_369_자동_운전 : BOOL; (* AT %MW87500.10 *) (* HOP_PBL_369_자동_운전 *)
    HOP_PBL_운전준비_ON : BOOL; (* AT %MW87500.0 *) (* HOP_PBL_운전준비_ON *)
    HOP_SSP_369_수동_선택 : BOOL; (* AT %MW87500.9 *) (* HOP_SSP_369_수동_선택 *)
    HOP_SSP_369_자동_선택 : BOOL; (* AT %MW87500.8 *) (* HOP_SSP_369_자동_선택 *)
    MCP_PBL_369_자동_운전 : BOOL; (* AT %MW87630.10 *) (* MCP PBL 369~-1 자동기동 *)
    MCP_PBL_운전준비_ON : BOOL; (* AT %MW87630.0 *) (* MCP_PBL_운전준비_ON *)
    MCP_SPB_작업완료_RESET : BOOL; (* AT %MW87631.6 *) (* MCP_SPB_작업완료_RESET *)
    MCP_SPB_작업완료_SET : BOOL; (* AT %MW87631.7 *) (* MCP_SPB_작업완료_SET *)
    MCP_SSP_369_수동_선택 : BOOL; (* AT %MW87630.8 *) (* MCP_SSP_369_수동_선택 *)
    MCP_SSP_369_자동_선택 : BOOL; (* AT %MW87630.9 *) (* MCP_SSP_369_자동_선택 *)
    R369_1_M_I_RB_3차_작업완료 : BOOL; (* AT %MW20081.4 *) (* R369_1_M_I_RB_3차_작업완료 *)
    R369_1_M_I_RB_간섭무_1 : BOOL; (* AT %MW20082.0 *) (* R369_1_M_I_RB_간섭무_1 *)
    R369_1_M_I_RB_원위치 : BOOL; (* AT %MW20080.3 *) (* R369_1_M_I_RB_원위치 *)
    R369_2_M_I_RB_2차_작업완료 : BOOL; (* AT %MW20091.3 *) (* R369_2_M_I_RB_2차_작업완료 *)
    R369_2_M_I_RB_간섭무_1 : BOOL; (* AT %MW20092.0 *) (* R369_2_M_I_RB_간섭무_1 *)
    R369_2_M_I_RB_원위치 : BOOL; (* AT %MW20090.3 *) (* R369_2_M_I_RB_원위치 *)
    S369_PHS_언로딩_이젝터_제품감지1 : BOOL; (* AT %MW86422.8 *) (* S369UD_PHS_AX_UD_제품감지_CHK1 *)
    S369_PHS_언로딩_이젝터_제품감지2 : BOOL; (* AT %MW86422.9 *) (* S369UD_PHS_AX_UD_제품감지_CHK2 *)
    S369_PRS_로딩_이젝터_LH_제품감지 : BOOL; (* AT %MW86412.1 *) (* S369LD_PRS_AX_LD_EJT_LH_CHK *)
    S369_PRS_로딩_이젝터_RH_제품감지 : BOOL; (* AT %MW86412.0 *) (* S369LD_PRS_AX_LD_EJT_RH_CHK *)
    S369_로딩버퍼_제품감지1 : BOOL; (* AT %MW86412.5 *) (* S369LD_LS_AX_CON_BELT_CHK1 *)
    S369_언로딩버퍼_제품감지1 : BOOL; (* AT %MW86422.5 *) (* S369UD_LS_AX_CON_BELT_CHK1 *)
    S369_이송버퍼01_제품감지1 : BOOL; (* AT %MW86422.6 *) (* S369UD_LS_AX_CON_BELT_CHK2 *)
    S369_이송버퍼02_제품감지1 : BOOL; (* AT %MW86422.7 *) (* S369UD_LS_AX_CON_BELT_CHK3 *)
    S369_이송버퍼03_제품감지1 : BOOL; (* AT %MW86412.7 *) (* S369LD_LS_AX_CON_BELT_CHK3 *)
    S369_이송버퍼04_제품감지1 : BOOL; (* AT %MW86412.6 *) (* S369LD_LS_AX_CON_BELT_CHK2 *)
END_VAR
VAR
    S369_READY : TON;
    T369_AUTO : TON;
END_VAR
VAR
    _t1 : BOOL;
    _t2 : BOOL;
    _t3 : BOOL;
    _t4 : BOOL;
    _t5 : BOOL;
    _t6 : BOOL;
END_VAR

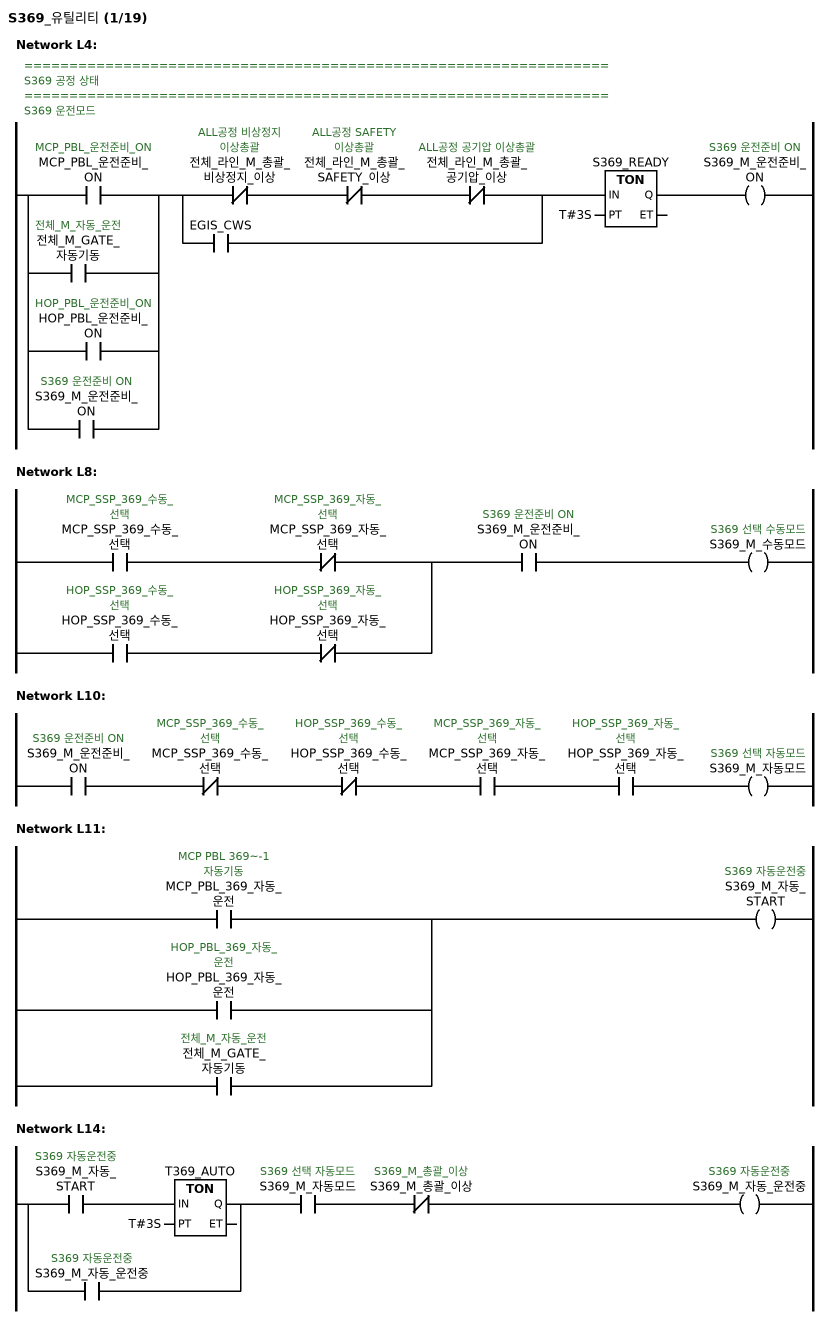
(* ================================================================= *)
(* S369 공정 상태 *)
(* ================================================================= *)
(* S369 운전모드 *)
(* Rung L4 *)
S369_READY(IN := (MCP_PBL_운전준비_ON OR 전체_M_GATE_자동기동 OR HOP_PBL_운전준비_ON OR S369_M_운전준비_ON) AND ((NOT 전체_라인_M_총괄_비상정지_이상 AND NOT 전체_라인_M_총괄_SAFETY_이상 AND NOT 전체_라인_M_총괄_공기압_이상) OR EGIS_CWS), PT := T#3S);
S369_M_운전준비_ON := S369_READY.Q;
(* Rung L8 *)
S369_M_수동모드 := ((MCP_SSP_369_수동_선택 AND NOT MCP_SSP_369_자동_선택) OR (HOP_SSP_369_수동_선택 AND NOT HOP_SSP_369_자동_선택)) AND S369_M_운전준비_ON;
(* Rung L10 *)
S369_M_자동모드 := S369_M_운전준비_ON AND NOT MCP_SSP_369_수동_선택 AND NOT HOP_SSP_369_수동_선택 AND MCP_SSP_369_자동_선택 AND HOP_SSP_369_자동_선택;
(* Rung L11 *)
S369_M_자동_START := MCP_PBL_369_자동_운전 OR HOP_PBL_369_자동_운전 OR 전체_M_GATE_자동기동;
(* Rung L14 *)
T369_AUTO(IN := S369_M_자동_START, PT := T#3S);
S369_M_자동_운전중 := (T369_AUTO.Q OR S369_M_자동_운전중) AND S369_M_자동모드 AND NOT S369_M_총괄_이상;

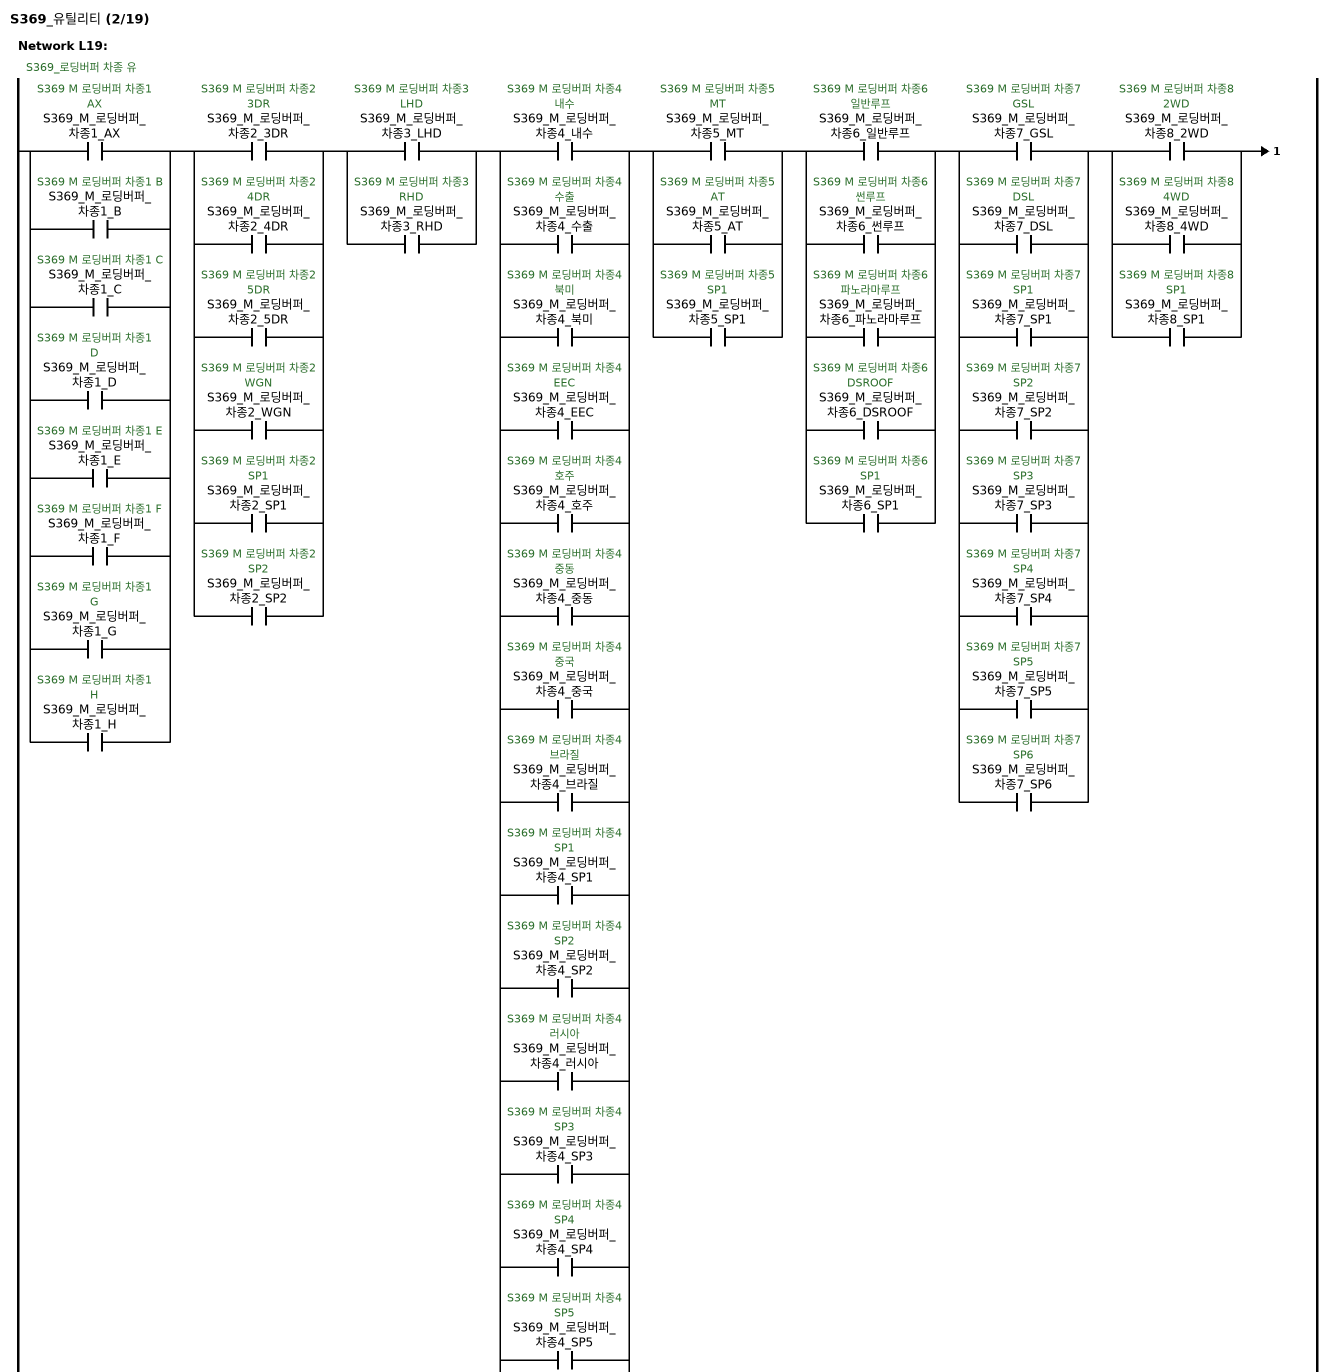

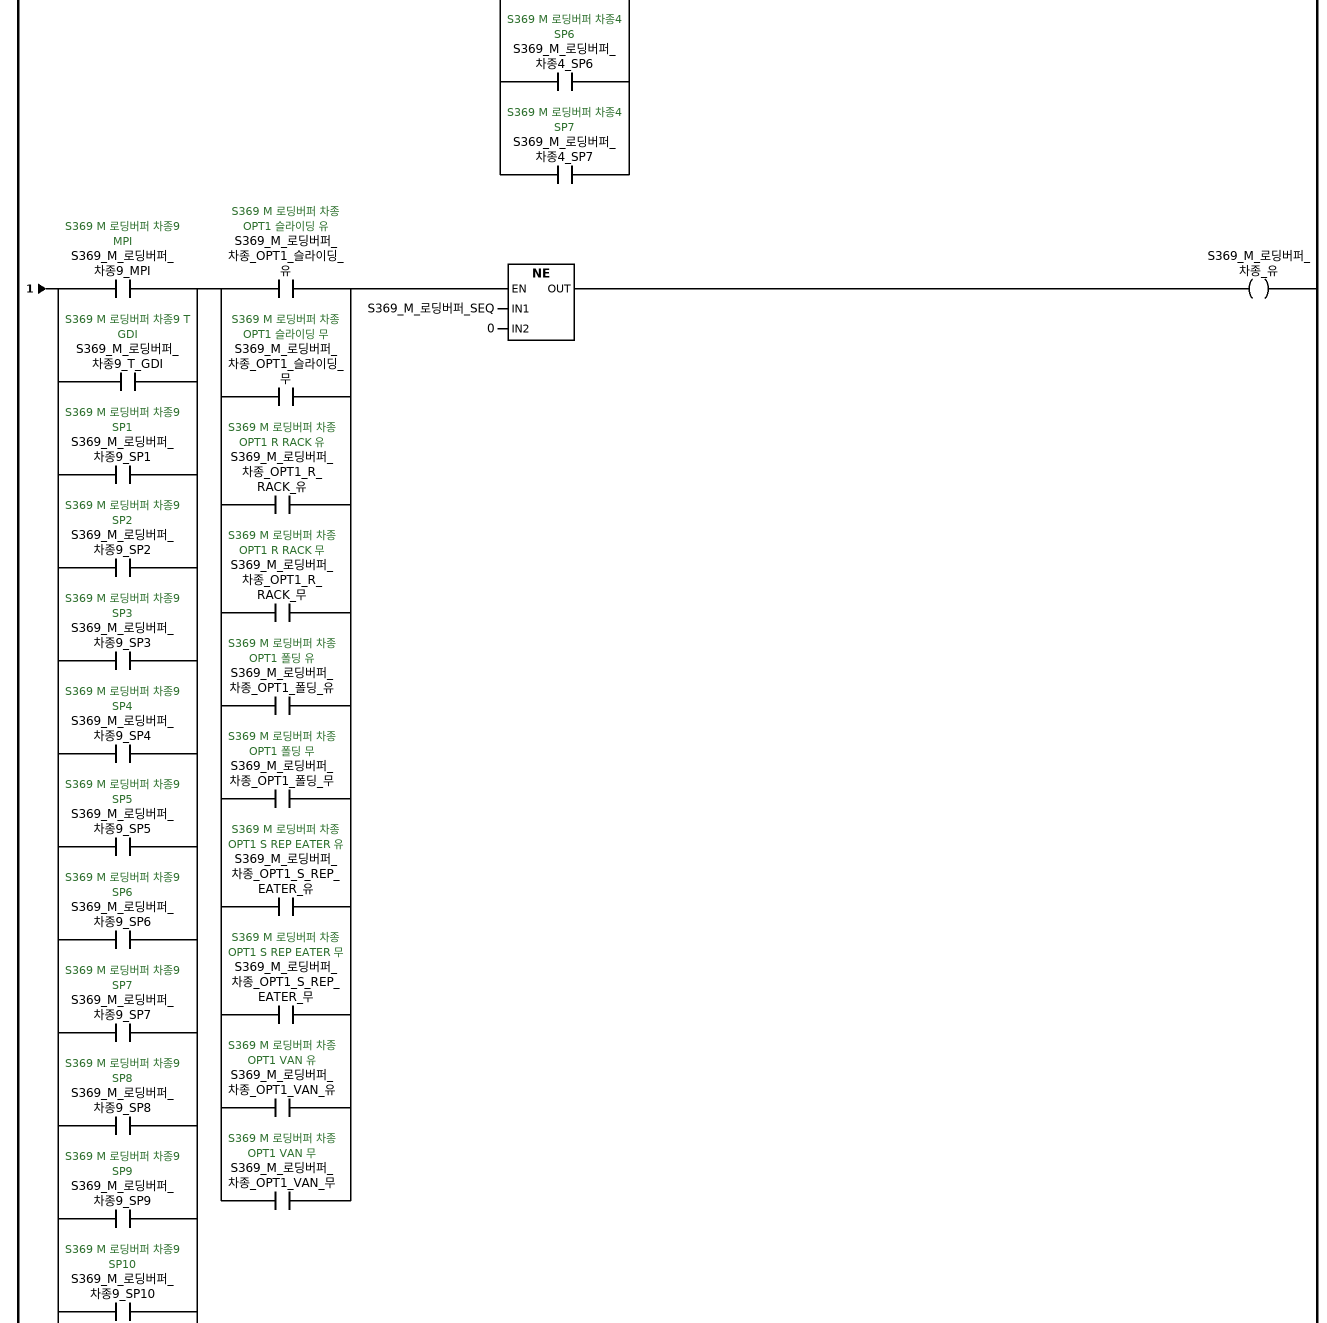

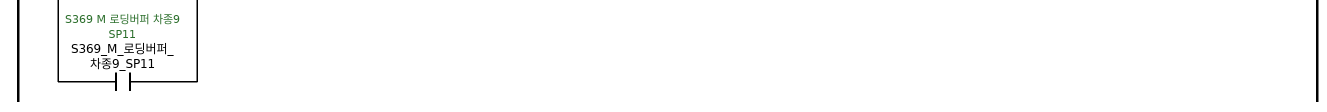
(* S369_로딩버퍼 차종 유 *)
(* Rung L19 *)
IF (S369_M_로딩버퍼_차종1_AX OR S369_M_로딩버퍼_차종1_B OR S369_M_로딩버퍼_차종1_C OR S369_M_로딩버퍼_차종1_D OR S369_M_로딩버퍼_차종1_E OR S369_M_로딩버퍼_차종1_F OR S369_M_로딩버퍼_차종1_G OR S369_M_로딩버퍼_차종1_H) AND (S369_M_로딩버퍼_차종2_3DR OR S369_M_로딩버퍼_차종2_4DR OR S369_M_로딩버퍼_차종2_5DR OR S369_M_로딩버퍼_차종2_WGN OR S369_M_로딩버퍼_차종2_SP1 OR S369_M_로딩버퍼_차종2_SP2) AND (S369_M_로딩버퍼_차종3_LHD OR S369_M_로딩버퍼_차종3_RHD) AND (S369_M_로딩버퍼_차종4_내수 OR S369_M_로딩버퍼_차종4_수출 OR S369_M_로딩버퍼_차종4_북미 OR S369_M_로딩버퍼_차종4_EEC OR S369_M_로딩버퍼_차종4_호주 OR S369_M_로딩버퍼_차종4_중동 OR S369_M_로딩버퍼_차종4_중국 OR S369_M_로딩버퍼_차종4_브라질 OR S369_M_로딩버퍼_차종4_SP1 OR S369_M_로딩버퍼_차종4_SP2 OR S369_M_로딩버퍼_차종4_러시아 OR S369_M_로딩버퍼_차종4_SP3 OR S369_M_로딩버퍼_차종4_SP4 OR S369_M_로딩버퍼_차종4_SP5 OR S369_M_로딩버퍼_차종4_SP6 OR S369_M_로딩버퍼_차종4_SP7) AND (S369_M_로딩버퍼_차종5_MT OR S369_M_로딩버퍼_차종5_AT OR S369_M_로딩버퍼_차종5_SP1) AND (S369_M_로딩버퍼_차종6_일반루프 OR S369_M_로딩버퍼_차종6_썬루프 OR S369_M_로딩버퍼_차종6_파노라마루프 OR S369_M_로딩버퍼_차종6_DSROOF OR S369_M_로딩버퍼_차종6_SP1) AND (S369_M_로딩버퍼_차종7_GSL OR S369_M_로딩버퍼_차종7_DSL OR S369_M_로딩버퍼_차종7_SP1 OR S369_M_로딩버퍼_차종7_SP2 OR S369_M_로딩버퍼_차종7_SP3 OR S369_M_로딩버퍼_차종7_SP4 OR S369_M_로딩버퍼_차종7_SP5 OR S369_M_로딩버퍼_차종7_SP6) AND (S369_M_로딩버퍼_차종8_2WD OR S369_M_로딩버퍼_차종8_4WD OR S369_M_로딩버퍼_차종8_SP1) AND (S369_M_로딩버퍼_차종9_MPI OR S369_M_로딩버퍼_차종9_T_GDI OR S369_M_로딩버퍼_차종9_SP1 OR S369_M_로딩버퍼_차종9_SP2 OR S369_M_로딩버퍼_차종9_SP3 OR S369_M_로딩버퍼_차종9_SP4 OR S369_M_로딩버퍼_차종9_SP5 OR S369_M_로딩버퍼_차종9_SP6 OR S369_M_로딩버퍼_차종9_SP7 OR S369_M_로딩버퍼_차종9_SP8 OR S369_M_로딩버퍼_차종9_SP9 OR S369_M_로딩버퍼_차종9_SP10 OR S369_M_로딩버퍼_차종9_SP11) AND (S369_M_로딩버퍼_차종_OPT1_슬라이딩_유 OR S369_M_로딩버퍼_차종_OPT1_슬라이딩_무 OR S369_M_로딩버퍼_차종_OPT1_R_RACK_유 OR S369_M_로딩버퍼_차종_OPT1_R_RACK_무 OR S369_M_로딩버퍼_차종_OPT1_폴딩_유 OR S369_M_로딩버퍼_차종_OPT1_폴딩_무 OR S369_M_로딩버퍼_차종_OPT1_S_REP_EATER_유 OR S369_M_로딩버퍼_차종_OPT1_S_REP_EATER_무 OR S369_M_로딩버퍼_차종_OPT1_VAN_유 OR S369_M_로딩버퍼_차종_OPT1_VAN_무) THEN
    _t1 := S369_M_로딩버퍼_SEQ <> 0;
END_IF;
S369_M_로딩버퍼_차종_유 := _t1;

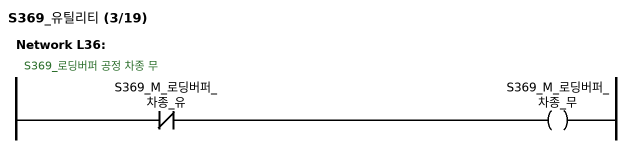
(* S369_로딩버퍼 공정 차종 무 *)
(* Rung L36 *)
S369_M_로딩버퍼_차종_무 := NOT S369_M_로딩버퍼_차종_유;

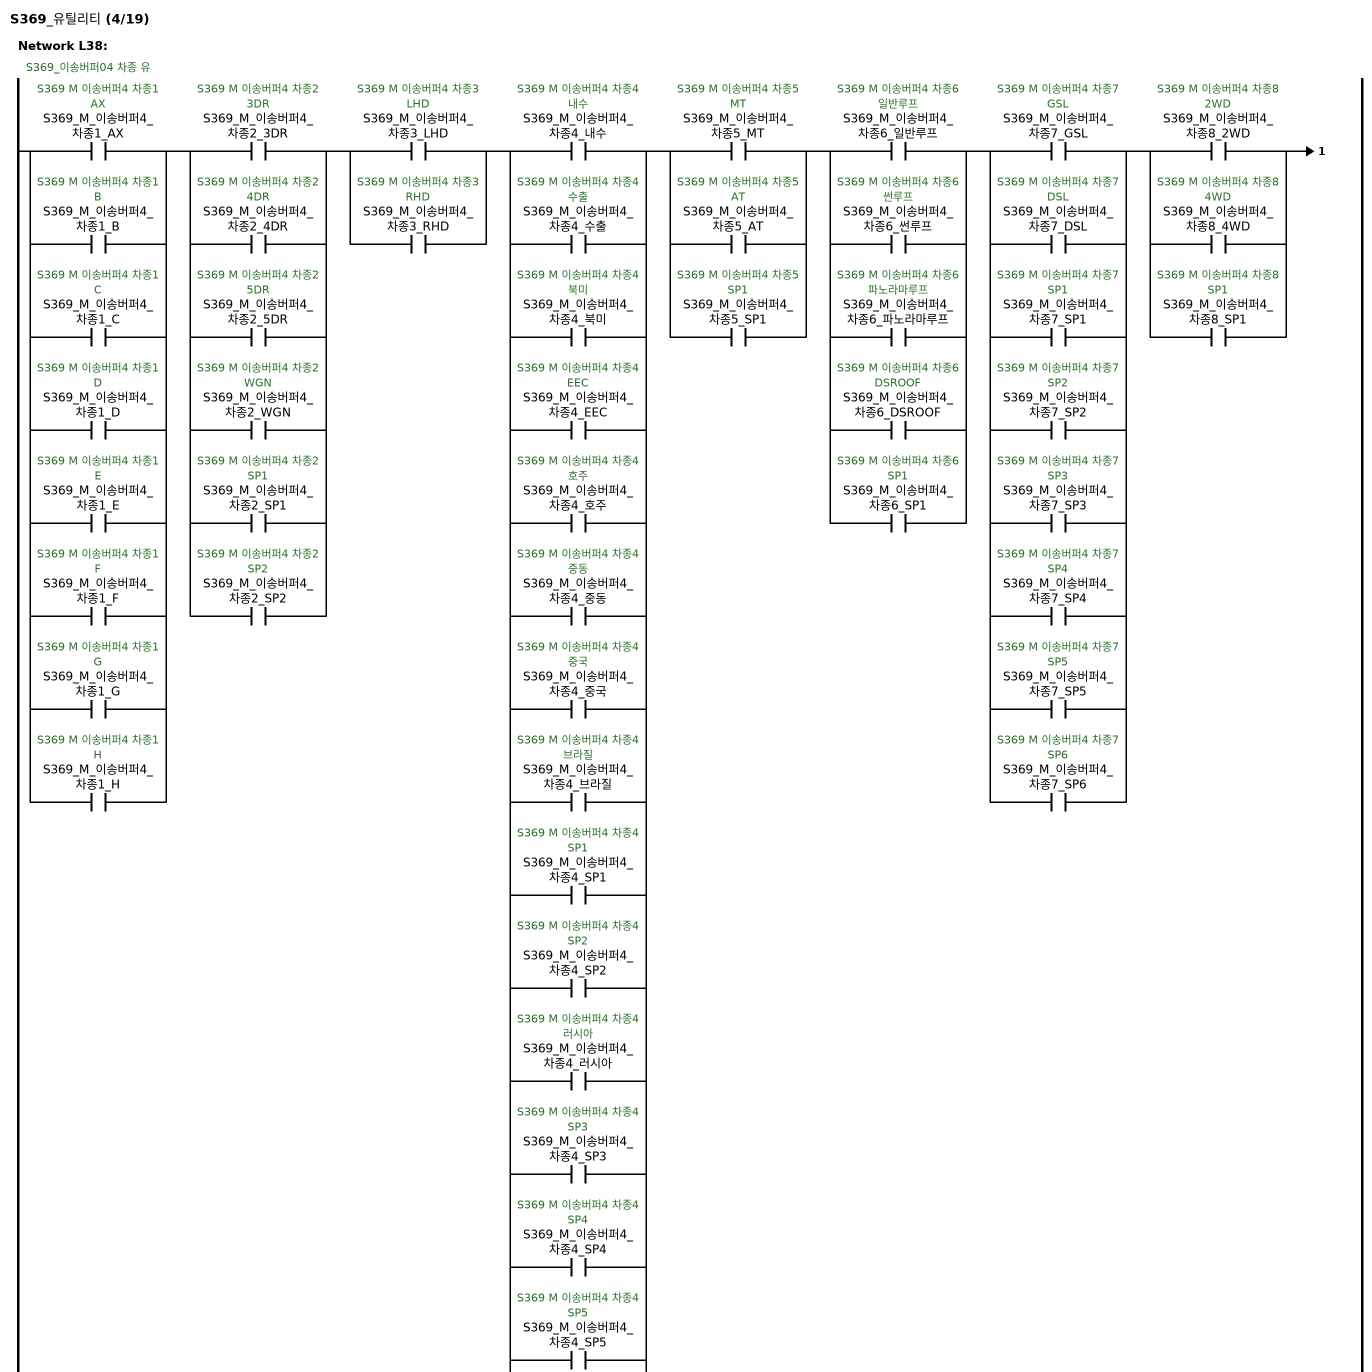

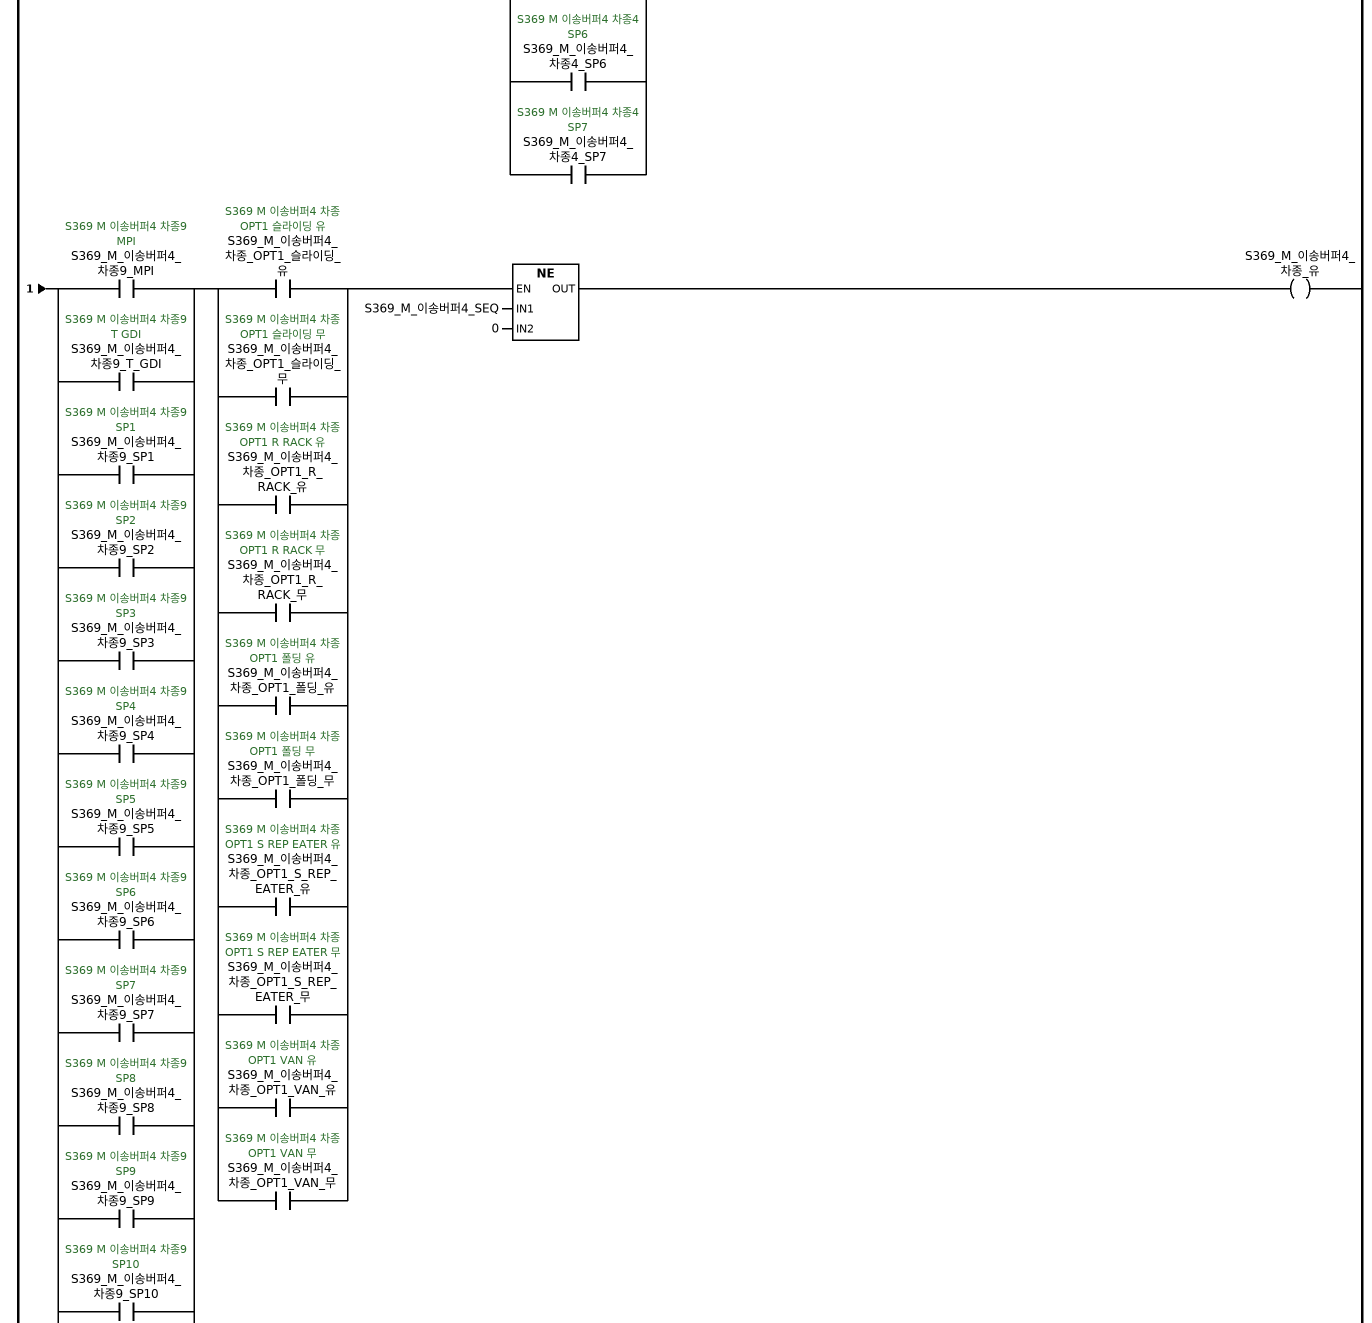

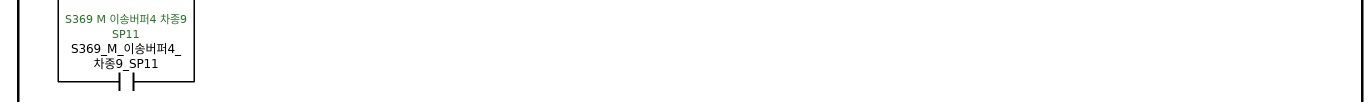
(* S369_이송버퍼04 차종 유 *)
(* Rung L38 *)
IF (S369_M_이송버퍼4_차종1_AX OR S369_M_이송버퍼4_차종1_B OR S369_M_이송버퍼4_차종1_C OR S369_M_이송버퍼4_차종1_D OR S369_M_이송버퍼4_차종1_E OR S369_M_이송버퍼4_차종1_F OR S369_M_이송버퍼4_차종1_G OR S369_M_이송버퍼4_차종1_H) AND (S369_M_이송버퍼4_차종2_3DR OR S369_M_이송버퍼4_차종2_4DR OR S369_M_이송버퍼4_차종2_5DR OR S369_M_이송버퍼4_차종2_WGN OR S369_M_이송버퍼4_차종2_SP1 OR S369_M_이송버퍼4_차종2_SP2) AND (S369_M_이송버퍼4_차종3_LHD OR S369_M_이송버퍼4_차종3_RHD) AND (S369_M_이송버퍼4_차종4_내수 OR S369_M_이송버퍼4_차종4_수출 OR S369_M_이송버퍼4_차종4_북미 OR S369_M_이송버퍼4_차종4_EEC OR S369_M_이송버퍼4_차종4_호주 OR S369_M_이송버퍼4_차종4_중동 OR S369_M_이송버퍼4_차종4_중국 OR S369_M_이송버퍼4_차종4_브라질 OR S369_M_이송버퍼4_차종4_SP1 OR S369_M_이송버퍼4_차종4_SP2 OR S369_M_이송버퍼4_차종4_러시아 OR S369_M_이송버퍼4_차종4_SP3 OR S369_M_이송버퍼4_차종4_SP4 OR S369_M_이송버퍼4_차종4_SP5 OR S369_M_이송버퍼4_차종4_SP6 OR S369_M_이송버퍼4_차종4_SP7) AND (S369_M_이송버퍼4_차종5_MT OR S369_M_이송버퍼4_차종5_AT OR S369_M_이송버퍼4_차종5_SP1) AND (S369_M_이송버퍼4_차종6_일반루프 OR S369_M_이송버퍼4_차종6_썬루프 OR S369_M_이송버퍼4_차종6_파노라마루프 OR S369_M_이송버퍼4_차종6_DSROOF OR S369_M_이송버퍼4_차종6_SP1) AND (S369_M_이송버퍼4_차종7_GSL OR S369_M_이송버퍼4_차종7_DSL OR S369_M_이송버퍼4_차종7_SP1 OR S369_M_이송버퍼4_차종7_SP2 OR S369_M_이송버퍼4_차종7_SP3 OR S369_M_이송버퍼4_차종7_SP4 OR S369_M_이송버퍼4_차종7_SP5 OR S369_M_이송버퍼4_차종7_SP6) AND (S369_M_이송버퍼4_차종8_2WD OR S369_M_이송버퍼4_차종8_4WD OR S369_M_이송버퍼4_차종8_SP1) AND (S369_M_이송버퍼4_차종9_MPI OR S369_M_이송버퍼4_차종9_T_GDI OR S369_M_이송버퍼4_차종9_SP1 OR S369_M_이송버퍼4_차종9_SP2 OR S369_M_이송버퍼4_차종9_SP3 OR S369_M_이송버퍼4_차종9_SP4 OR S369_M_이송버퍼4_차종9_SP5 OR S369_M_이송버퍼4_차종9_SP6 OR S369_M_이송버퍼4_차종9_SP7 OR S369_M_이송버퍼4_차종9_SP8 OR S369_M_이송버퍼4_차종9_SP9 OR S369_M_이송버퍼4_차종9_SP10 OR S369_M_이송버퍼4_차종9_SP11) AND (S369_M_이송버퍼4_차종_OPT1_슬라이딩_유 OR S369_M_이송버퍼4_차종_OPT1_슬라이딩_무 OR S369_M_이송버퍼4_차종_OPT1_R_RACK_유 OR S369_M_이송버퍼4_차종_OPT1_R_RACK_무 OR S369_M_이송버퍼4_차종_OPT1_폴딩_유 OR S369_M_이송버퍼4_차종_OPT1_폴딩_무 OR S369_M_이송버퍼4_차종_OPT1_S_REP_EATER_유 OR S369_M_이송버퍼4_차종_OPT1_S_REP_EATER_무 OR S369_M_이송버퍼4_차종_OPT1_VAN_유 OR S369_M_이송버퍼4_차종_OPT1_VAN_무) THEN
    _t2 := S369_M_이송버퍼4_SEQ <> 0;
END_IF;
S369_M_이송버퍼4_차종_유 := _t2;

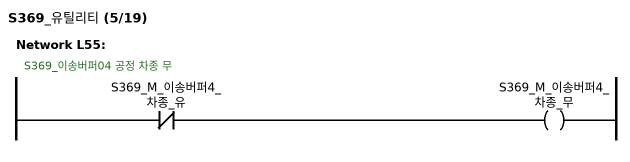
(* S369_이송버퍼04 공정 차종 무 *)
(* Rung L55 *)
S369_M_이송버퍼4_차종_무 := NOT S369_M_이송버퍼4_차종_유;

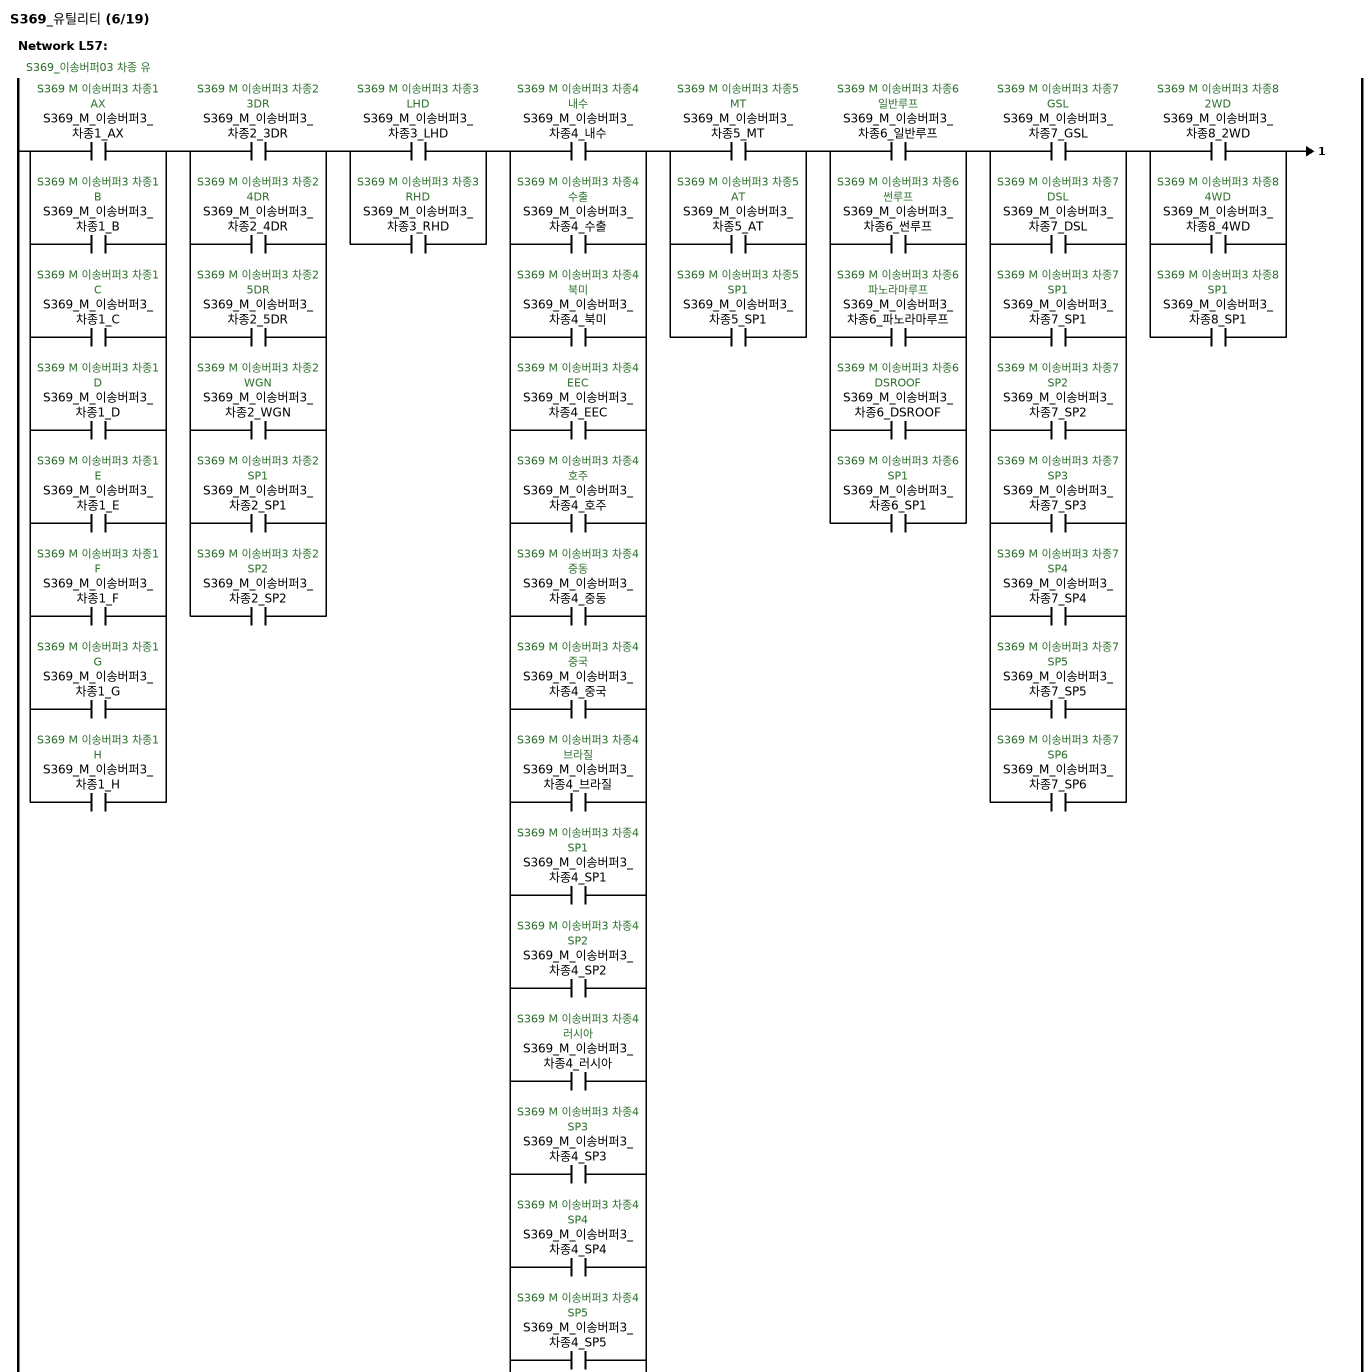

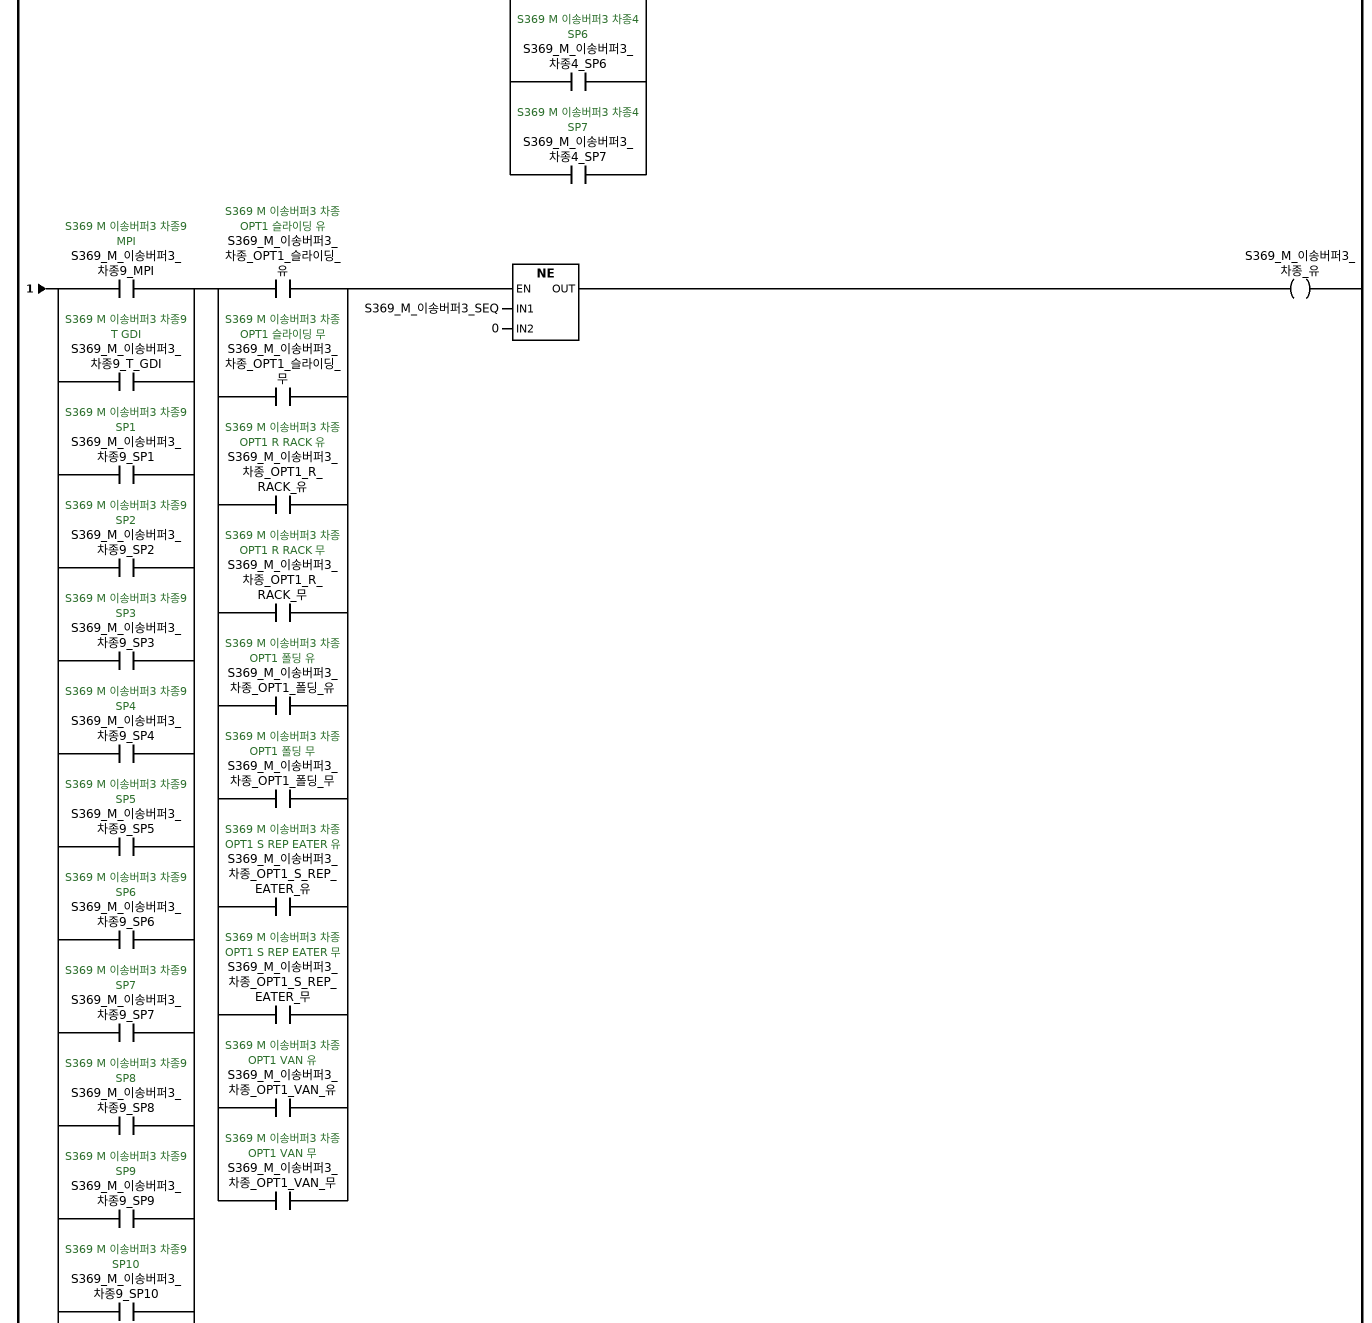

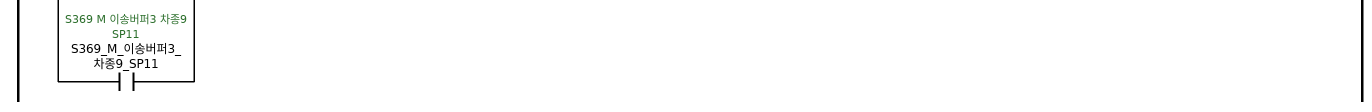
(* S369_이송버퍼03 차종 유 *)
(* Rung L57 *)
IF (S369_M_이송버퍼3_차종1_AX OR S369_M_이송버퍼3_차종1_B OR S369_M_이송버퍼3_차종1_C OR S369_M_이송버퍼3_차종1_D OR S369_M_이송버퍼3_차종1_E OR S369_M_이송버퍼3_차종1_F OR S369_M_이송버퍼3_차종1_G OR S369_M_이송버퍼3_차종1_H) AND (S369_M_이송버퍼3_차종2_3DR OR S369_M_이송버퍼3_차종2_4DR OR S369_M_이송버퍼3_차종2_5DR OR S369_M_이송버퍼3_차종2_WGN OR S369_M_이송버퍼3_차종2_SP1 OR S369_M_이송버퍼3_차종2_SP2) AND (S369_M_이송버퍼3_차종3_LHD OR S369_M_이송버퍼3_차종3_RHD) AND (S369_M_이송버퍼3_차종4_내수 OR S369_M_이송버퍼3_차종4_수출 OR S369_M_이송버퍼3_차종4_북미 OR S369_M_이송버퍼3_차종4_EEC OR S369_M_이송버퍼3_차종4_호주 OR S369_M_이송버퍼3_차종4_중동 OR S369_M_이송버퍼3_차종4_중국 OR S369_M_이송버퍼3_차종4_브라질 OR S369_M_이송버퍼3_차종4_SP1 OR S369_M_이송버퍼3_차종4_SP2 OR S369_M_이송버퍼3_차종4_러시아 OR S369_M_이송버퍼3_차종4_SP3 OR S369_M_이송버퍼3_차종4_SP4 OR S369_M_이송버퍼3_차종4_SP5 OR S369_M_이송버퍼3_차종4_SP6 OR S369_M_이송버퍼3_차종4_SP7) AND (S369_M_이송버퍼3_차종5_MT OR S369_M_이송버퍼3_차종5_AT OR S369_M_이송버퍼3_차종5_SP1) AND (S369_M_이송버퍼3_차종6_일반루프 OR S369_M_이송버퍼3_차종6_썬루프 OR S369_M_이송버퍼3_차종6_파노라마루프 OR S369_M_이송버퍼3_차종6_DSROOF OR S369_M_이송버퍼3_차종6_SP1) AND (S369_M_이송버퍼3_차종7_GSL OR S369_M_이송버퍼3_차종7_DSL OR S369_M_이송버퍼3_차종7_SP1 OR S369_M_이송버퍼3_차종7_SP2 OR S369_M_이송버퍼3_차종7_SP3 OR S369_M_이송버퍼3_차종7_SP4 OR S369_M_이송버퍼3_차종7_SP5 OR S369_M_이송버퍼3_차종7_SP6) AND (S369_M_이송버퍼3_차종8_2WD OR S369_M_이송버퍼3_차종8_4WD OR S369_M_이송버퍼3_차종8_SP1) AND (S369_M_이송버퍼3_차종9_MPI OR S369_M_이송버퍼3_차종9_T_GDI OR S369_M_이송버퍼3_차종9_SP1 OR S369_M_이송버퍼3_차종9_SP2 OR S369_M_이송버퍼3_차종9_SP3 OR S369_M_이송버퍼3_차종9_SP4 OR S369_M_이송버퍼3_차종9_SP5 OR S369_M_이송버퍼3_차종9_SP6 OR S369_M_이송버퍼3_차종9_SP7 OR S369_M_이송버퍼3_차종9_SP8 OR S369_M_이송버퍼3_차종9_SP9 OR S369_M_이송버퍼3_차종9_SP10 OR S369_M_이송버퍼3_차종9_SP11) AND (S369_M_이송버퍼3_차종_OPT1_슬라이딩_유 OR S369_M_이송버퍼3_차종_OPT1_슬라이딩_무 OR S369_M_이송버퍼3_차종_OPT1_R_RACK_유 OR S369_M_이송버퍼3_차종_OPT1_R_RACK_무 OR S369_M_이송버퍼3_차종_OPT1_폴딩_유 OR S369_M_이송버퍼3_차종_OPT1_폴딩_무 OR S369_M_이송버퍼3_차종_OPT1_S_REP_EATER_유 OR S369_M_이송버퍼3_차종_OPT1_S_REP_EATER_무 OR S369_M_이송버퍼3_차종_OPT1_VAN_유 OR S369_M_이송버퍼3_차종_OPT1_VAN_무) THEN
    _t3 := S369_M_이송버퍼3_SEQ <> 0;
END_IF;
S369_M_이송버퍼3_차종_유 := _t3;

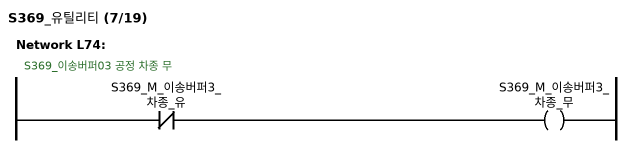
(* S369_이송버퍼03 공정 차종 무 *)
(* Rung L74 *)
S369_M_이송버퍼3_차종_무 := NOT S369_M_이송버퍼3_차종_유;

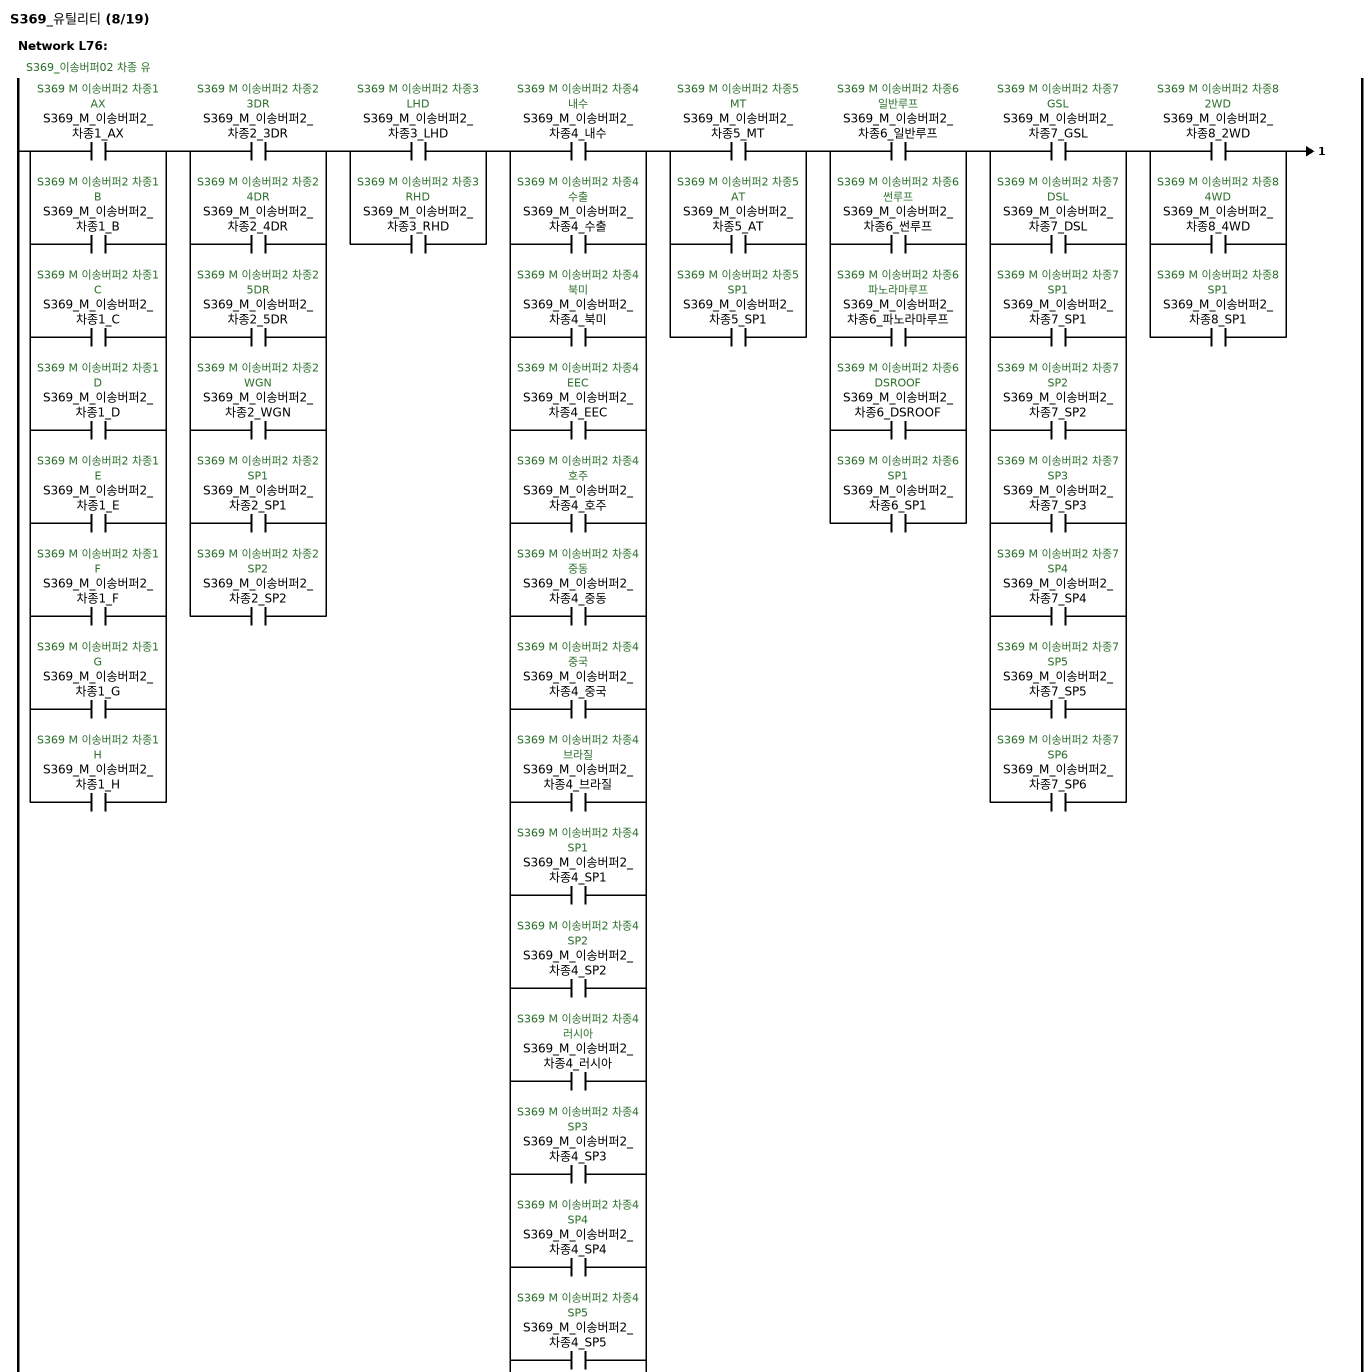

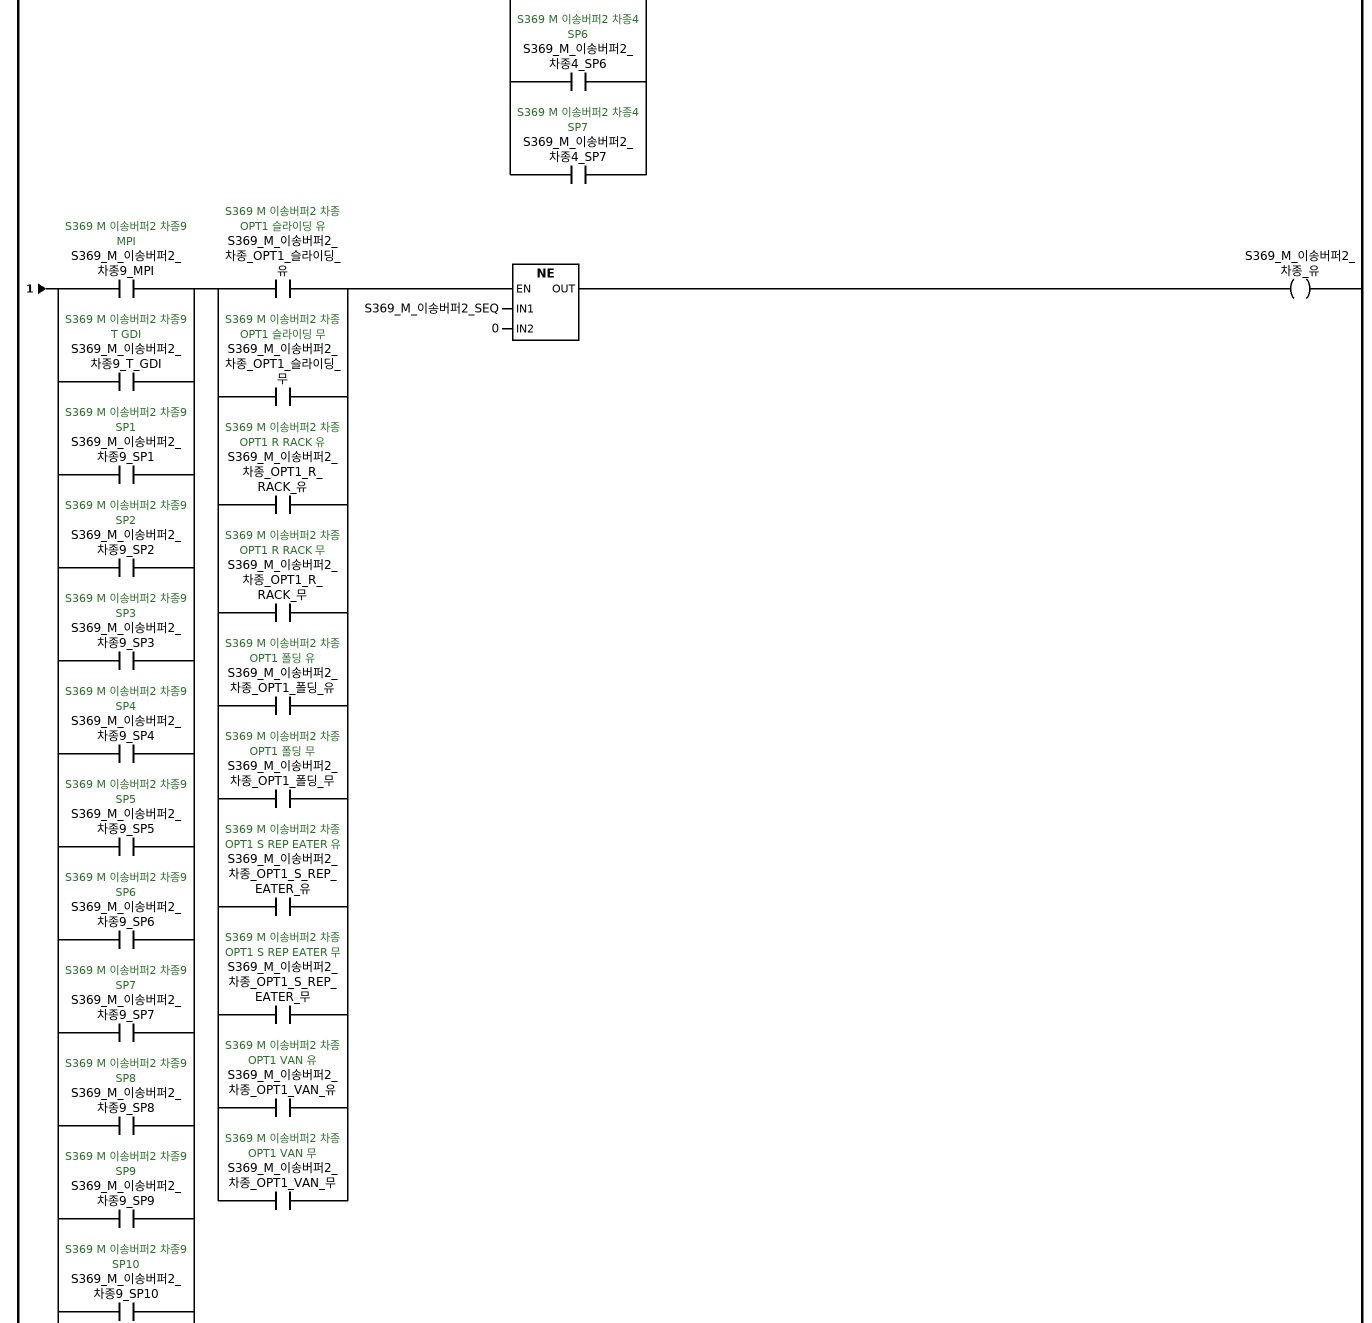

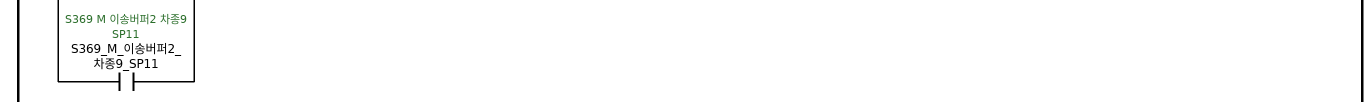
(* S369_이송버퍼02 차종 유 *)
(* Rung L76 *)
IF (S369_M_이송버퍼2_차종1_AX OR S369_M_이송버퍼2_차종1_B OR S369_M_이송버퍼2_차종1_C OR S369_M_이송버퍼2_차종1_D OR S369_M_이송버퍼2_차종1_E OR S369_M_이송버퍼2_차종1_F OR S369_M_이송버퍼2_차종1_G OR S369_M_이송버퍼2_차종1_H) AND (S369_M_이송버퍼2_차종2_3DR OR S369_M_이송버퍼2_차종2_4DR OR S369_M_이송버퍼2_차종2_5DR OR S369_M_이송버퍼2_차종2_WGN OR S369_M_이송버퍼2_차종2_SP1 OR S369_M_이송버퍼2_차종2_SP2) AND (S369_M_이송버퍼2_차종3_LHD OR S369_M_이송버퍼2_차종3_RHD) AND (S369_M_이송버퍼2_차종4_내수 OR S369_M_이송버퍼2_차종4_수출 OR S369_M_이송버퍼2_차종4_북미 OR S369_M_이송버퍼2_차종4_EEC OR S369_M_이송버퍼2_차종4_호주 OR S369_M_이송버퍼2_차종4_중동 OR S369_M_이송버퍼2_차종4_중국 OR S369_M_이송버퍼2_차종4_브라질 OR S369_M_이송버퍼2_차종4_SP1 OR S369_M_이송버퍼2_차종4_SP2 OR S369_M_이송버퍼2_차종4_러시아 OR S369_M_이송버퍼2_차종4_SP3 OR S369_M_이송버퍼2_차종4_SP4 OR S369_M_이송버퍼2_차종4_SP5 OR S369_M_이송버퍼2_차종4_SP6 OR S369_M_이송버퍼2_차종4_SP7) AND (S369_M_이송버퍼2_차종5_MT OR S369_M_이송버퍼2_차종5_AT OR S369_M_이송버퍼2_차종5_SP1) AND (S369_M_이송버퍼2_차종6_일반루프 OR S369_M_이송버퍼2_차종6_썬루프 OR S369_M_이송버퍼2_차종6_파노라마루프 OR S369_M_이송버퍼2_차종6_DSROOF OR S369_M_이송버퍼2_차종6_SP1) AND (S369_M_이송버퍼2_차종7_GSL OR S369_M_이송버퍼2_차종7_DSL OR S369_M_이송버퍼2_차종7_SP1 OR S369_M_이송버퍼2_차종7_SP2 OR S369_M_이송버퍼2_차종7_SP3 OR S369_M_이송버퍼2_차종7_SP4 OR S369_M_이송버퍼2_차종7_SP5 OR S369_M_이송버퍼2_차종7_SP6) AND (S369_M_이송버퍼2_차종8_2WD OR S369_M_이송버퍼2_차종8_4WD OR S369_M_이송버퍼2_차종8_SP1) AND (S369_M_이송버퍼2_차종9_MPI OR S369_M_이송버퍼2_차종9_T_GDI OR S369_M_이송버퍼2_차종9_SP1 OR S369_M_이송버퍼2_차종9_SP2 OR S369_M_이송버퍼2_차종9_SP3 OR S369_M_이송버퍼2_차종9_SP4 OR S369_M_이송버퍼2_차종9_SP5 OR S369_M_이송버퍼2_차종9_SP6 OR S369_M_이송버퍼2_차종9_SP7 OR S369_M_이송버퍼2_차종9_SP8 OR S369_M_이송버퍼2_차종9_SP9 OR S369_M_이송버퍼2_차종9_SP10 OR S369_M_이송버퍼2_차종9_SP11) AND (S369_M_이송버퍼2_차종_OPT1_슬라이딩_유 OR S369_M_이송버퍼2_차종_OPT1_슬라이딩_무 OR S369_M_이송버퍼2_차종_OPT1_R_RACK_유 OR S369_M_이송버퍼2_차종_OPT1_R_RACK_무 OR S369_M_이송버퍼2_차종_OPT1_폴딩_유 OR S369_M_이송버퍼2_차종_OPT1_폴딩_무 OR S369_M_이송버퍼2_차종_OPT1_S_REP_EATER_유 OR S369_M_이송버퍼2_차종_OPT1_S_REP_EATER_무 OR S369_M_이송버퍼2_차종_OPT1_VAN_유 OR S369_M_이송버퍼2_차종_OPT1_VAN_무) THEN
    _t4 := S369_M_이송버퍼2_SEQ <> 0;
END_IF;
S369_M_이송버퍼2_차종_유 := _t4;

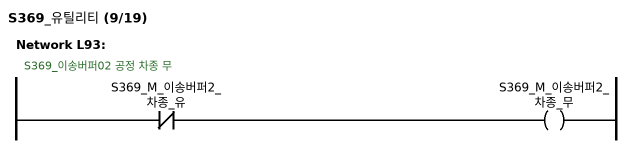
(* S369_이송버퍼02 공정 차종 무 *)
(* Rung L93 *)
S369_M_이송버퍼2_차종_무 := NOT S369_M_이송버퍼2_차종_유;

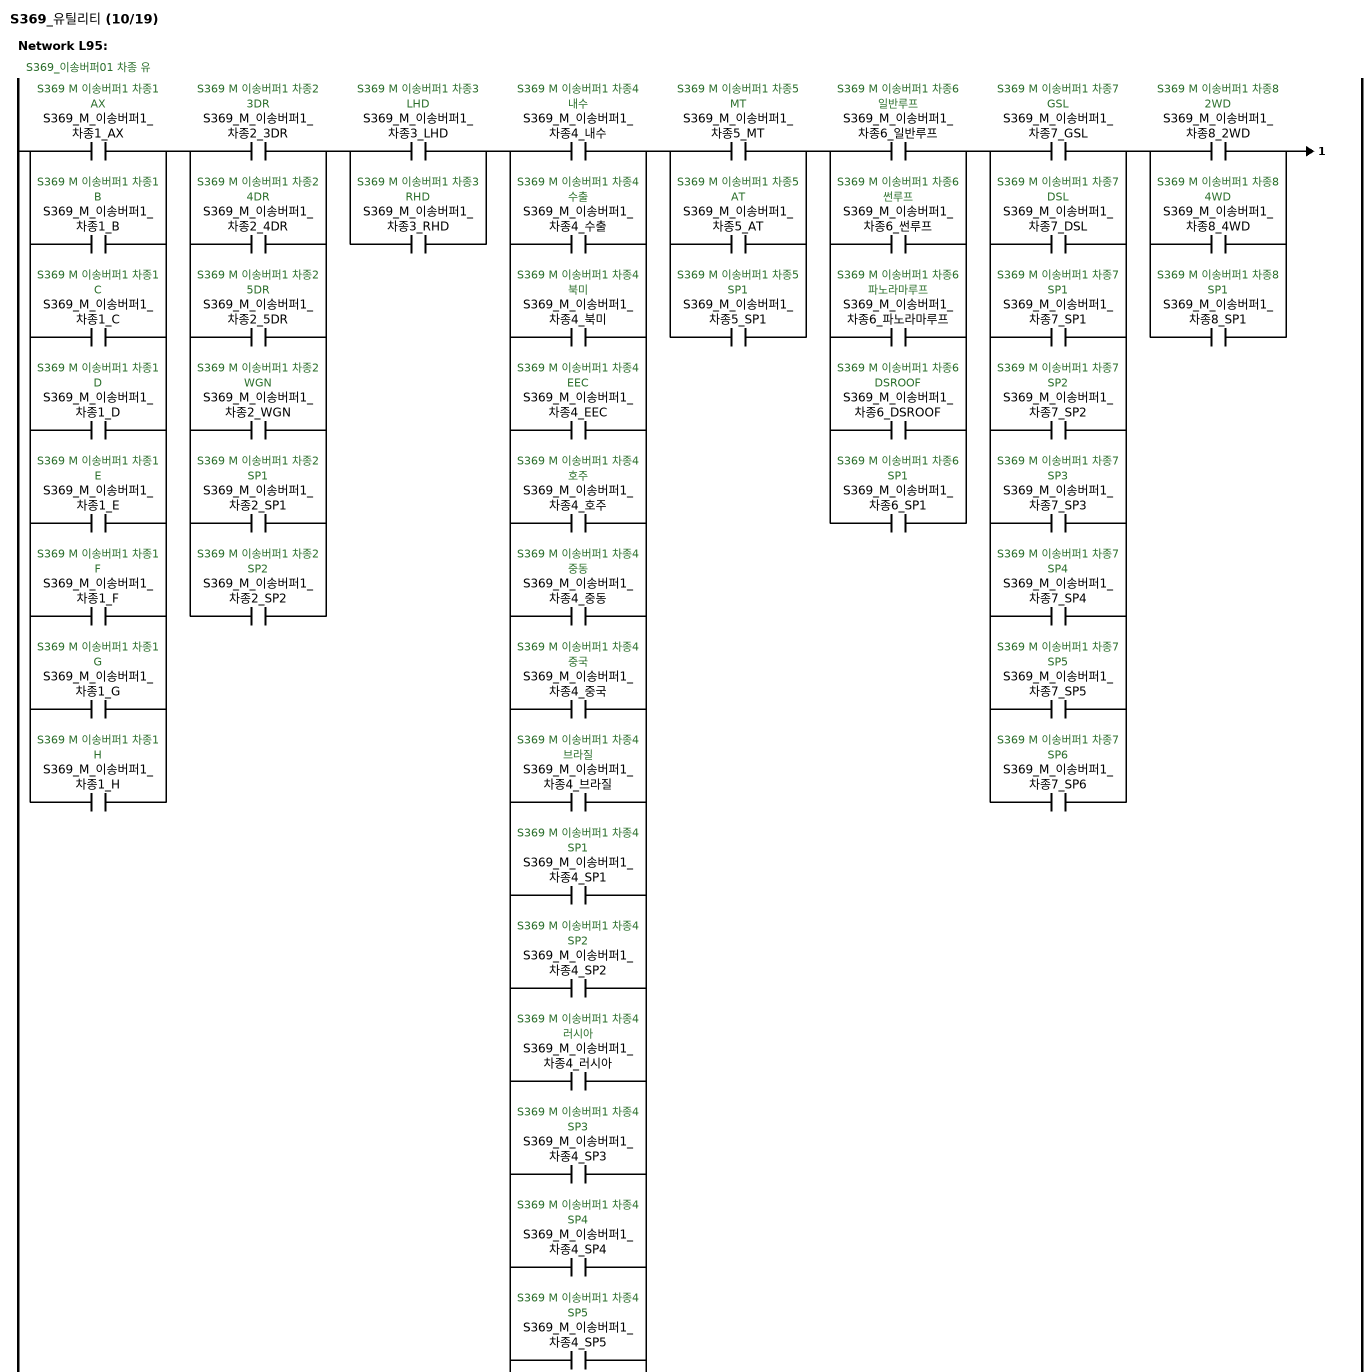
(* [picture p286: S369_유틸리티 rungs L95-L95] *)

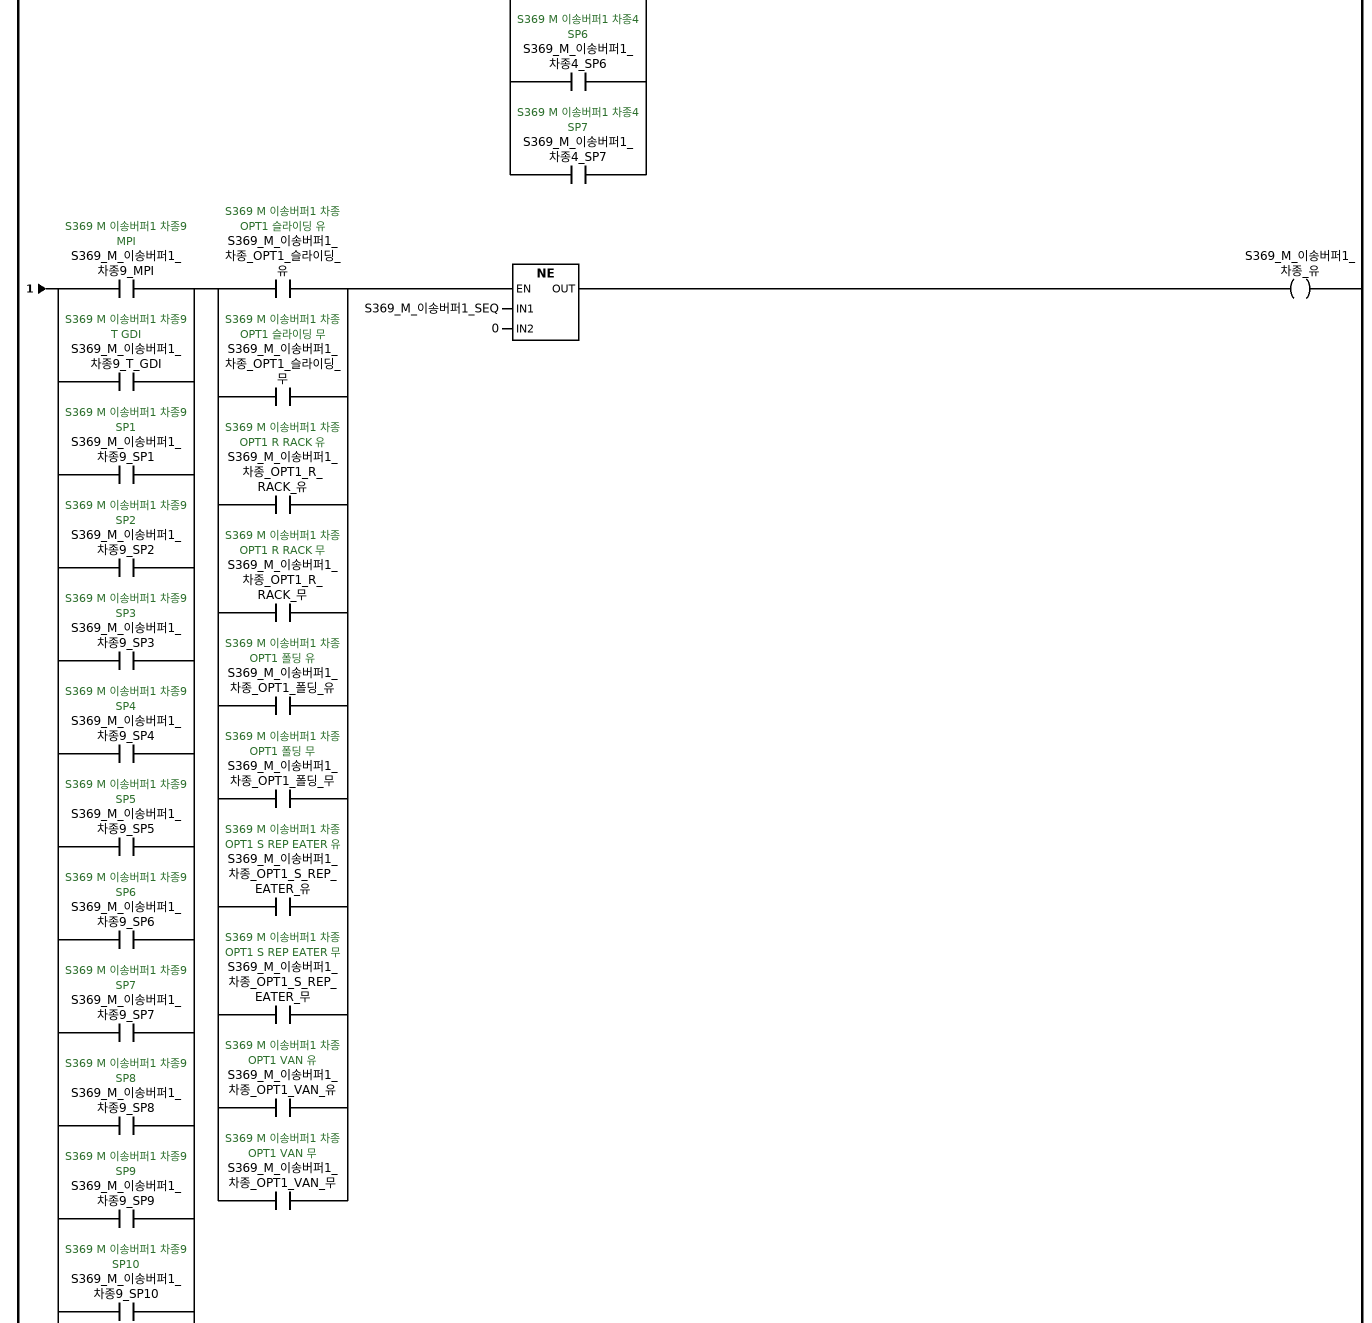

